  [343] = "19.57,-101.88,1.00,-90.00,-68.25,0.00,0,"
  [344] = "19.49,-101.70,1.00,-90.00,-68.30,0.00,1,"
  [345] = "19.42,-101.51,1.00,-90.00,-68.34,0.00,0,"
  [346] = "19.35,-101.32,1.00,-90.00,-68.38,0.00,1,"
  [347] = "19.27,-101.14,1.00,-90.00,-68.42,0.00,0,"
  [348] = "19.20,-100.95,1.00,-90.00,-68.46,0.00,1,"
  [349] = "19.13,-100.77,1.00,-90.00,-68.50,0.00,0,"
  [350] = "19.05,-100.58,1.00,-90.00,-68.55,0.00,1,"
  [351] = "18.98,-100.39,1.00,-90.00,-68.59,0.00,0,"
  [352] = "18.91,-100.21,1.00,-90.00,-68.63,0.00,1,"
  [353] = "18.83,-100.02,1.00,-90.00,-68.67,0.00,0,"
  [354] = "18.76,-99.83,1.00,-90.00,-68.71,0.00,1,"
  [355] = "18.69,-99.65,1.00,-90.00,-68.75,0.00,0,"
  [356] = "18.62,-99.46,1.00,-90.00,-68.80,0.00,1,"
  [357] = "18.54,-99.28,1.00,-90.00,-68.84,0.00,0,"
  [358] = "18.47,-99.09,1.00,-90.00,-68.88,0.00,1,"
  [359] = "18.40,-98.90,1.00,-90.00,-68.92,0.00,0,"
  [360] = "18.33,-98.72,1.00,-90.00,-68.96,0.00,1,"
  [361] = "18.26,-98.53,1.00,-90.00,-69.00,0.00,0,"
  [362] = "18.19,-98.34,1.00,-90.00,-69.05,0.00,1,"
  [363] = "18.11,-98.16,1.00,-90.00,-69.09,0.00,0,"
  [364] = "18.04,-97.97,1.00,-90.00,-69.13,0.00,1,"
  [365] = "17.97,-97.78,1.00,-90.00,-69.17,0.00,0,"
  [366] = "17.90,-97.59,1.00,-90.00,-69.21,0.00,1,"
  [367] = "17.83,-97.41,1.00,-90.00,-69.25,0.00,0,"
  [368] = "17.76,-97.22,1.00,-90.00,-69.30,0.00,1,"
  [369] = "17.69,-97.03,1.00,-90.00,-69.34,0.00,0,"
  [370] = "17.62,-96.85,1.00,-90.00,-69.38,0.00,1,"
  [371] = "17.55,-96.66,1.00,-90.00,-69.42,0.00,0,"
  [372] = "17.48,-96.47,1.00,-90.00,-69.46,0.00,1,"
  [373] = "17.41,-96.28,1.00,-90.00,-69.50,0.00,0,"
  [374] = "17.34,-96.10,1.00,-90.00,-69.55,0.00,1,"
  [375] = "17.27,-95.91,1.00,-90.00,-69.59,0.00,0,"
  [376] = "17.20,-95.72,1.00,-90.00,-69.63,0.00,1,"
  [377] = "17.13,-95.53,1.00,-90.00,-69.67,0.00,0,"
  [378] = "17.06,-95.35,1.00,-90.00,-69.71,0.00,1,"
  [379] = "16.99,-95.16,1.00,-90.00,-69.75,0.00,0,"
  [380] = "16.92,-94.97,1.00,-90.00,-69.80,0.00,1,"
  [381] = "16.85,-94.78,1.00,-90.00,-69.84,0.00,0,"
  [382] = "16.78,-94.60,1.00,-90.00,-69.88,0.00,1,"
  [383] = "16.71,-94.41,1.00,-90.00,-69.92,0.00,0,"
  [384] = "16.64,-94.22,1.00,-90.00,-69.96,0.00,1,"
  [385] = "16.58,-94.03,1.00,-90.00,-70.01,0.00,0,"
  [386] = "16.51,-93.84,1.00,-90.00,-70.05,0.00,1,"
  [387] = "16.44,-93.66,1.00,-90.00,-70.09,0.00,0,"
  [388] = "16.37,-93.47,1.00,-90.00,-70.13,0.00,1,"
  [389] = "16.30,-93.28,1.00,-90.00,-70.17,0.00,0,"
  [390] = "16.24,-93.09,1.00,-90.00,-70.21,0.00,1,"
  [391] = "16.17,-92.90,1.00,-90.00,-70.26,0.00,0,"
  [392] = "16.10,-92.72,1.00,-90.00,-70.30,0.00,1,"
  [393] = "16.03,-92.53,1.00,-90.00,-70.34,0.00,0,"
  [394] = "15.97,-92.34,1.00,-90.00,-70.38,0.00,1,"
  [395] = "15.90,-92.15,1.00,-90.00,-70.42,0.00,0,"
  [396] = "15.83,-91.96,1.00,-90.00,-70.46,0.00,1,"
  [397] = "15.77,-91.77,1.00,-90.00,-70.50,0.00,0,"
  [398] = "15.70,-91.59,1.00,-90.00,-70.55,0.00,1,"
  [399] = "15.63,-91.40,1.00,-90.00,-70.59,0.00,0,"
  [400] = "15.57,-91.21,1.00,-90.00,-70.63,0.00,1,"
  [401] = "15.50,-91.02,1.00,-90.00,-70.67,0.00,0,"
  [402] = "15.43,-90.83,1.00,-90.00,-70.71,0.00,1,"
  [403] = "15.37,-90.64,1.00,-90.00,-70.76,0.00,0,"
  [404] = "15.30,-90.45,1.00,-90.00,-70.80,0.00,1,"
  [405] = "15.24,-90.26,1.00,-90.00,-70.84,0.00,0,"
  [406] = "15.17,-90.08,1.00,-90.00,-70.88,0.00,1,"
  [407] = "15.10,-89.89,1.00,-90.00,-70.92,0.00,0,"
  [408] = "15.04,-89.70,1.00,-90.00,-70.96,0.00,1,"
  [409] = "14.97,-89.51,1.00,-90.00,-71.01,0.00,0,"
  [410] = "14.91,-89.32,1.00,-90.00,-71.05,0.00,1,"
  [411] = "14.84,-89.13,1.00,-90.00,-71.09,0.00,0,"
  [412] = "14.78,-88.94,1.00,-90.00,-71.13,0.00,1,"
  [413] = "14.72,-88.75,1.00,-90.00,-71.17,0.00,0,"
  [414] = "14.65,-88.56,1.00,-90.00,-71.21,0.00,1,"
  [415] = "14.59,-88.37,1.00,-90.00,-71.26,0.00,0,"
  [416] = "14.52,-88.18,1.00,-90.00,-71.30,0.00,1,"
  [417] = "14.46,-87.99,1.00,-90.00,-71.34,0.00,0,"
  [418] = "14.39,-87.80,1.00,-90.00,-71.38,0.00,1,"
  [419] = "14.33,-87.61,1.00,-90.00,-71.42,0.00,0,"
  [420] = "14.27,-87.43,1.00,-90.00,-71.46,0.00,1,"
  [421] = "14.20,-87.24,1.00,-90.00,-71.51,0.00,0,"
  [422] = "14.14,-87.05,1.00,-90.00,-71.55,0.00,1,"
  [423] = "14.08,-86.86,1.00,-90.00,-71.59,0.00,0,"
  [424] = "14.01,-86.67,1.00,-90.00,-71.63,0.00,1,"
  [425] = "13.95,-86.48,1.00,-90.00,-71.67,0.00,0,"
  [426] = "13.89,-86.29,1.00,-90.00,-71.71,0.00,1,"
  [427] = "13.82,-86.10,1.00,-90.00,-71.76,0.00,0,"
  [428] = "13.76,-85.91,1.00,-90.00,-71.80,0.00,1,"
  [429] = "13.70,-85.72,1.00,-90.00,-71.84,0.00,0,"
  [430] = "13.64,-85.53,1.00,-90.00,-71.88,0.00,1,"
  [431] = "13.58,-85.34,1.00,-90.00,-71.92,0.00,0,"
  [432] = "13.51,-85.15,1.00,-90.00,-71.96,0.00,1,"
  [433] = "13.45,-84.96,1.00,-90.00,-72.01,0.00,0,"
  [434] = "13.39,-84.77,1.00,-90.00,-72.05,0.00,1,"
  [435] = "13.33,-84.58,1.00,-90.00,-72.09,0.00,0,"
  [436] = "13.27,-84.39,1.00,-90.00,-72.13,0.00,1,"
  [437] = "13.21,-84.19,1.00,-90.00,-72.17,0.00,0,"
  [438] = "13.14,-84.00,1.00,-90.00,-72.21,0.00,1,"
  [439] = "13.08,-83.81,1.00,-90.00,-72.26,0.00,0,"
  [440] = "13.02,-83.62,1.00,-90.00,-72.30,0.00,1,"
  [441] = "12.96,-83.43,1.00,-90.00,-72.34,0.00,0,"
  [442] = "12.90,-83.24,1.00,-90.00,-72.38,0.00,1,"
  [443] = "12.84,-83.05,1.00,-90.00,-72.42,0.00,0,"
  [444] = "12.78,-82.86,1.00,-90.00,-72.46,0.00,1,"
  [445] = "12.72,-82.67,1.00,-90.00,-72.51,0.00,0,"
  [446] = "12.66,-82.48,1.00,-90.00,-72.55,0.00,1,"
  [447] = "12.60,-82.29,1.00,-90.00,-72.59,0.00,0,"
  [448] = "12.54,-82.10,1.00,-90.00,-72.63,0.00,1,"
  [449] = "12.48,-81.91,1.00,-90.00,-72.67,0.00,0,"
  [450] = "12.42,-81.72,1.00,-90.00,-72.71,0.00,1,"
  [451] = "12.36,-81.52,1.00,-90.00,-72.76,0.00,0,"
  [452] = "12.30,-81.33,1.00,-90.00,-72.80,0.00,1,"
  [453] = "12.24,-81.14,1.00,-90.00,-72.84,0.00,0,"
  [454] = "12.18,-80.95,1.00,-90.00,-72.88,0.00,1,"
  [455] = "12.13,-80.76,1.00,-90.00,-72.92,0.00,0,"
  [456] = "12.07,-80.57,1.00,-90.00,-72.96,0.00,1,"
  [457] = "12.01,-80.38,1.00,-90.00,-73.01,0.00,0,"
  [458] = "11.95,-80.19,1.00,-90.00,-73.05,0.00,1,"
  [459] = "11.89,-80.00,1.00,-90.00,-73.09,0.00,0,"
  [460] = "11.83,-79.80,1.00,-90.00,-73.13,0.00,1,"
  [461] = "11.78,-79.61,1.00,-90.00,-73.17,0.00,0,"
  [462] = "11.72,-79.42,1.00,-90.00,-73.21,0.00,1,"
  [463] = "11.66,-79.23,1.00,-90.00,-73.26,0.00,0,"
  [464] = "11.60,-79.04,1.00,-90.00,-73.30,0.00,1,"
  [465] = "11.55,-78.85,1.00,-90.00,-73.34,0.00,0,"
  [466] = "11.49,-78.66,1.00,-90.00,-73.38,0.00,1,"
  [467] = "11.43,-78.46,1.00,-90.00,-73.42,0.00,0,"
  [468] = "11.37,-78.27,1.00,-90.00,-73.46,0.00,1,"
  [469] = "11.32,-78.08,1.00,-90.00,-73.51,0.00,0,"
  [470] = "11.26,-77.89,1.00,-90.00,-73.55,0.00,1,"
  [471] = "11.20,-77.70,1.00,-90.00,-73.59,0.00,0,"
  [472] = "11.15,-77.50,1.00,-90.00,-73.63,0.00,1,"
  [473] = "11.09,-77.31,1.00,-90.00,-73.67,0.00,0,"
  [474] = "11.04,-77.12,1.00,-90.00,-73.71,0.00,1,"
  [475] = "10.98,-76.93,1.00,-90.00,-73.76,0.00,0,"
  [476] = "10.92,-76.74,1.00,-90.00,-73.80,0.00,1,"
  [477] = "10.87,-76.54,1.00,-90.00,-73.84,0.00,0,"
  [478] = "10.81,-76.35,1.00,-90.00,-73.88,0.00,1,"
  [479] = "10.76,-76.16,1.00,-90.00,-73.92,0.00,0,"
  [480] = "10.70,-75.97,1.00,-90.00,-73.96,0.00,1,"
  [481] = "10.65,-75.78,1.00,-90.00,-74.01,0.00,0,"
  [482] = "10.59,-75.58,1.00,-90.00,-74.05,0.00,1,"
  [483] = "10.54,-75.39,1.00,-90.00,-74.09,0.00,0,"
  [484] = "10.48,-75.20,1.00,-90.00,-74.13,0.00,1,"
  [485] = "10.43,-75.01,1.00,-90.00,-74.17,0.00,0,"
  [486] = "10.37,-74.81,1.00,-90.00,-74.21,0.00,1,"
  [487] = "10.32,-74.62,1.00,-90.00,-74.26,0.00,0,"
  [488] = "10.26,-74.43,1.00,-90.00,-74.30,0.00,1,"
  [489] = "10.21,-74.24,1.00,-90.00,-74.34,0.00,0,"
  [490] = "10.16,-74.04,1.00,-90.00,-74.38,0.00,1,"
  [491] = "10.10,-73.85,1.00,-90.00,-74.42,0.00,0,"
  [492] = "10.05,-73.66,1.00,-90.00,-74.46,0.00,1,"
  [493] = "9.99,-73.47,1.00,-90.00,-74.51,0.00,0,"
  [494] = "9.94,-73.27,1.00,-90.00,-74.55,0.00,1,"
  [495] = "9.89,-73.08,1.00,-90.00,-74.59,0.00,0,"
  [496] = "9.84,-72.89,1.00,-90.00,-74.63,0.00,1,"
  [497] = "9.78,-72.69,1.00,-90.00,-74.67,0.00,0,"
  [498] = "9.73,-72.50,1.00,-90.00,-74.71,0.00,1,"
  [499] = "9.68,-72.31,1.00,-90.00,-74.76,0.00,0,"
  [500] = "9.62,-72.12,1.00,-90.00,-74.80,0.00,1,"
  [501] = "9.57,-71.92,1.00,-90.00,-74.84,0.00,0,"
  [502] = "9.52,-71.73,1.00,-90.00,-74.88,0.00,1,"
  [503] = "9.47,-71.54,1.00,-90.00,-74.92,0.00,0,"
  [504] = "9.42,-71.34,1.00,-90.00,-74.96,0.00,1,"
  [505] = "9.36,-71.15,1.00,-90.00,-75.01,0.00,0,"
  [506] = "9.31,-70.96,1.00,-90.00,-75.05,0.00,1,"
  [507] = "9.26,-70.76,1.00,-90.00,-75.09,0.00,0,"
  [508] = "9.21,-70.57,1.00,-90.00,-75.13,0.00,1,"
  [509] = "9.16,-70.38,1.00,-90.00,-75.17,0.00,0,"
  [510] = "9.11,-70.18,1.00,-90.00,-75.21,0.00,1,"
  [511] = "9.06,-69.99,1.00,-90.00,-75.26,0.00,0,"
  [512] = "9.00,-69.80,1.00,-90.00,-75.30,0.00,1,"
  [513] = "8.95,-69.60,1.00,-90.00,-75.34,0.00,0,"
  [514] = "8.90,-69.41,1.00,-90.00,-75.38,0.00,1,"
  [515] = "8.85,-69.22,1.00,-90.00,-75.42,0.00,0,"
  [516] = "8.80,-69.02,1.00,-90.00,-75.46,0.00,1,"
  [517] = "8.75,-68.83,1.00,-90.00,-75.51,0.00,0,"
  [518] = "8.70,-68.64,1.00,-90.00,-75.55,0.00,1,"
  [519] = "8.65,-68.44,1.00,-90.00,-75.59,0.00,0,"
  [520] = "8.60,-68.25,1.00,-90.00,-75.63,0.00,1,"
  [521] = "8.55,-68.05,1.00,-90.00,-75.67,0.00,0,"
  [522] = "8.50,-67.86,1.00,-90.00,-75.71,0.00,1,"
  [523] = "8.46,-67.67,1.00,-90.00,-75.76,0.00,0,"
  [524] = "8.41,-67.47,1.00,-90.00,-75.80,0.00,1,"
  [525] = "8.36,-67.28,1.00,-90.00,-75.84,0.00,0,"
  [526] = "8.31,-67.09,1.00,-90.00,-75.88,0.00,1,"
  [527] = "8.26,-66.89,1.00,-90.00,-75.92,0.00,0,"
  [528] = "8.21,-66.70,1.00,-90.00,-75.96,0.00,1,"
  [529] = "8.16,-66.50,1.00,-90.00,-76.01,0.00,0,"
  [530] = "8.11,-66.31,1.00,-90.00,-76.05,0.00,1,"
  [531] = "8.07,-66.11,1.00,-90.00,-76.09,0.00,0,"
  [532] = "8.02,-65.92,1.00,-90.00,-76.13,0.00,1,"
  [533] = "7.97,-65.73,1.00,-90.00,-76.17,0.00,0,"
  [534] = "7.92,-65.53,1.00,-90.00,-76.21,0.00,1,"
  [535] = "7.87,-65.34,1.00,-90.00,-76.26,0.00,0,"
  [536] = "7.83,-65.14,1.00,-90.00,-76.30,0.00,1,"
  [537] = "7.78,-64.95,1.00,-90.00,-76.34,0.00,0,"
  [538] = "7.73,-64.76,1.00,-90.00,-76.38,0.00,1,"
  [539] = "7.69,-64.56,1.00,-90.00,-76.42,0.00,0,"
  [540] = "7.64,-64.37,1.00,-90.00,-76.46,0.00,1,"
  [541] = "7.59,-64.17,1.00,-90.00,-76.51,0.00,0,"
  [542] = "7.55,-63.98,1.00,-90.00,-76.55,0.00,1,"
  [543] = "7.50,-63.78,1.00,-90.00,-76.59,0.00,0,"
  [544] = "7.45,-63.59,1.00,-90.00,-76.63,0.00,1,"
  [545] = "7.41,-63.39,1.00,-90.00,-76.67,0.00,0,"
  [546] = "7.36,-63.20,1.00,-90.00,-76.71,0.00,1,"
  [547] = "7.31,-63.00,1.00,-90.00,-76.76,0.00,0,"
  [548] = "7.27,-62.81,1.00,-90.00,-76.80,0.00,1,"
  [549] = "7.22,-62.61,1.00,-90.00,-76.84,0.00,0,"
  [550] = "7.18,-62.42,1.00,-90.00,-76.88,0.00,1,"
  [551] = "7.13,-62.23,1.00,-90.00,-76.92,0.00,0,"
  [552] = "7.09,-62.03,1.00,-90.00,-76.96,0.00,1,"
  [553] = "7.04,-61.84,1.00,-90.00,-77.01,0.00,0,"
  [554] = "7.00,-61.64,1.00,-90.00,-77.05,0.00,1,"
  [555] = "6.95,-61.45,1.00,-90.00,-77.09,0.00,0,"
  [556] = "6.91,-61.25,1.00,-90.00,-77.13,0.00,1,"
  [557] = "6.86,-61.06,1.00,-90.00,-77.17,0.00,0,"
  [558] = "6.82,-60.86,1.00,-90.00,-77.21,0.00,1,"
  [559] = "6.77,-60.67,1.00,-90.00,-77.26,0.00,0,"
  [560] = "6.73,-60.47,1.00,-90.00,-77.30,0.00,1,"
  [561] = "6.69,-60.28,1.00,-90.00,-77.34,0.00,0,"
  [562] = "6.64,-60.08,1.00,-90.00,-77.38,0.00,1,"
  [563] = "6.60,-59.89,1.00,-90.00,-77.42,0.00,0,"
  [564] = "6.56,-59.69,1.00,-90.00,-77.46,0.00,1,"
  [565] = "6.51,-59.49,1.00,-90.00,-77.51,0.00,0,"
  [566] = "6.47,-59.30,1.00,-90.00,-77.55,0.00,1,"
  [567] = "6.43,-59.10,1.00,-90.00,-77.59,0.00,0,"
  [568] = "6.38,-58.91,1.00,-90.00,-77.63,0.00,1,"
  [569] = "6.34,-58.71,1.00,-90.00,-77.67,0.00,0,"
  [570] = "6.30,-58.52,1.00,-90.00,-77.71,0.00,1,"
  [571] = "6.26,-58.32,1.00,-90.00,-77.76,0.00,0,"
  [572] = "6.21,-58.13,1.00,-90.00,-77.80,0.00,1,"
  [573] = "6.17,-57.93,1.00,-90.00,-77.84,0.00,0,"
  [574] = "6.13,-57.74,1.00,-90.00,-77.88,0.00,1,"
  [575] = "6.09,-57.54,1.00,-90.00,-77.92,0.00,0,"
  [576] = "6.05,-57.35,1.00,-90.00,-77.96,0.00,1,"
  [577] = "6.00,-57.15,1.00,-90.00,-78.01,0.00,0,"
  [578] = "5.96,-56.95,1.00,-90.00,-78.05,0.00,1,"
  [579] = "5.92,-56.76,1.00,-90.00,-78.09,0.00,0,"
  [580] = "5.88,-56.56,1.00,-90.00,-78.13,0.00,1,"
  [581] = "5.84,-56.37,1.00,-90.00,-78.17,0.00,0,"
  [582] = "5.80,-56.17,1.00,-90.00,-78.21,0.00,1,"
  [583] = "5.76,-55.98,1.00,-90.00,-78.26,0.00,0,"
  [584] = "5.72,-55.78,1.00,-90.00,-78.30,0.00,1,"
  [585] = "5.68,-55.58,1.00,-90.00,-78.34,0.00,0,"
  [586] = "5.64,-55.39,1.00,-90.00,-78.38,0.00,1,"
  [587] = "5.60,-55.19,1.00,-90.00,-78.42,0.00,0,"
  [588] = "5.56,-55.00,1.00,-90.00,-78.46,0.00,1,"
  [589] = "5.52,-54.80,1.00,-90.00,-78.51,0.00,0,"
  [590] = "5.48,-54.60,1.00,-90.00,-78.55,0.00,1,"
  [591] = "5.44,-54.41,1.00,-90.00,-78.59,0.00,0,"
  [592] = "5.40,-54.21,1.00,-90.00,-78.63,0.00,1,"
  [593] = "5.36,-54.02,1.00,-90.00,-78.67,0.00,0,"
  [594] = "5.32,-53.82,1.00,-90.00,-78.71,0.00,1,"
  [595] = "5.28,-53.62,1.00,-90.00,-78.76,0.00,0,"
  [596] = "5.24,-53.43,1.00,-90.00,-78.80,0.00,1,"
  [597] = "5.20,-53.23,1.00,-90.00,-78.84,0.00,0,"
  [598] = "5.16,-53.03,1.00,-90.00,-78.88,0.00,1,"
  [599] = "5.12,-52.84,1.00,-90.00,-78.92,0.00,0,"
  [600] = "5.09,-52.64,1.00,-90.00,-78.96,0.00,1,"
  [601] = "5.05,-52.45,1.00,-90.00,-79.01,0.00,0,"
  [602] = "5.01,-52.25,1.00,-90.00,-79.05,0.00,1,"
  [603] = "4.97,-52.05,1.00,-90.00,-79.09,0.00,0,"
  [604] = "4.93,-51.86,1.00,-90.00,-79.13,0.00,1,"
  [605] = "4.90,-51.66,1.00,-90.00,-79.17,0.00,0,"
  [606] = "4.86,-51.46,1.00,-90.00,-79.21,0.00,1,"
  [607] = "4.82,-51.27,1.00,-90.00,-79.26,0.00,0,"
  [608] = "4.78,-51.07,1.00,-90.00,-79.30,0.00,1,"
  [609] = "4.75,-50.87,1.00,-90.00,-79.34,0.00,0,"
  [610] = "4.71,-50.68,1.00,-90.00,-79.38,0.00,1,"
  [611] = "4.67,-50.48,1.00,-90.00,-79.42,0.00,0,"
  [612] = "4.64,-50.28,1.00,-90.00,-79.46,0.00,1,"
  [613] = "4.60,-50.09,1.00,-90.00,-79.51,0.00,0,"
  [614] = "4.56,-49.89,1.00,-90.00,-79.55,0.00,1,"
  [615] = "4.53,-49.69,1.00,-90.00,-79.59,0.00,0,"
  [616] = "4.49,-49.50,1.00,-90.00,-79.63,0.00,1,"
  [617] = "4.46,-49.30,1.00,-90.00,-79.67,0.00,0,"
  [618] = "4.42,-49.10,1.00,-90.00,-79.71,0.00,1,"
  [619] = "4.38,-48.91,1.00,-90.00,-79.76,0.00,0,"
  [620] = "4.35,-48.71,1.00,-90.00,-79.80,0.00,1,"
  [621] = "4.31,-48.51,1.00,-90.00,-79.84,0.00,0,"
  [622] = "4.28,-48.32,1.00,-90.00,-79.88,0.00,1,"
  [623] = "4.24,-48.12,1.00,-90.00,-79.92,0.00,0,"
  [624] = "4.21,-47.92,1.00,-90.00,-79.96,0.00,1,"
  [625] = "4.17,-47.73,1.00,-90.00,-80.01,0.00,0,"
  [626] = "4.14,-47.53,1.00,-90.00,-80.05,0.00,1,"
  [627] = "4.10,-47.33,1.00,-90.00,-80.09,0.00,0,"
  [628] = "4.07,-47.14,1.00,-90.00,-80.13,0.00,1,"
  [629] = "4.04,-46.94,1.00,-90.00,-80.17,0.00,0,"
  [630] = "4.00,-46.74,1.00,-90.00,-80.21,0.00,1,"
  [631] = "3.97,-46.54,1.00,-90.00,-80.26,0.00,0,"
  [632] = "3.93,-46.35,1.00,-90.00,-80.30,0.00,1,"
  [633] = "3.90,-46.15,1.00,-90.00,-80.34,0.00,0,"
  [634] = "3.87,-45.95,1.00,-90.00,-80.38,0.00,1,"
  [635] = "3.83,-45.76,1.00,-90.00,-80.42,0.00,0,"
  [636] = "3.80,-45.56,1.00,-90.00,-80.46,0.00,1,"
  [637] = "3.77,-45.36,1.00,-90.00,-80.51,0.00,0,"
  [638] = "3.73,-45.16,1.00,-90.00,-80.55,0.00,1,"
  [639] = "3.70,-44.97,1.00,-90.00,-80.59,0.00,0,"
  [640] = "3.67,-44.77,1.00,-90.00,-80.63,0.00,1,"
  [641] = "3.64,-44.57,1.00,-90.00,-80.67,0.00,0,"
  [642] = "3.60,-44.37,1.00,-90.00,-80.71,0.00,1,"
  [643] = "3.57,-44.18,1.00,-90.00,-80.76,0.00,0,"
  [644] = "3.54,-43.98,1.00,-90.00,-80.80,0.00,1,"
  [645] = "3.51,-43.78,1.00,-90.00,-80.84,0.00,0,"
  [646] = "3.48,-43.58,1.00,-90.00,-80.88,0.00,1,"
  [647] = "3.44,-43.39,1.00,-90.00,-80.92,0.00,0,"
  [648] = "3.41,-43.19,1.00,-90.00,-80.96,0.00,1,"
  [649] = "3.38,-42.99,1.00,-90.00,-81.01,0.00,0,"
  [650] = "3.35,-42.79,1.00,-90.00,-81.05,0.00,1,"
  [651] = "3.32,-42.60,1.00,-90.00,-81.09,0.00,0,"
  [652] = "3.29,-42.40,1.00,-90.00,-81.13,0.00,1,"
  [653] = "3.26,-42.20,1.00,-90.00,-81.17,0.00,0,"
  [654] = "3.23,-42.00,1.00,-90.00,-81.21,0.00,1,"
  [655] = "3.20,-41.81,1.00,-90.00,-81.26,0.00,0,"
  [656] = "3.17,-41.61,1.00,-90.00,-81.30,0.00,1,"
  [657] = "3.14,-41.41,1.00,-90.00,-81.34,0.00,0,"
  [658] = "3.11,-41.21,1.00,-90.00,-81.38,0.00,1,"
  [659] = "3.08,-41.02,1.00,-90.00,-81.42,0.00,0,"
  [660] = "3.05,-40.82,1.00,-90.00,-81.46,0.00,1,"
  [661] = "3.02,-40.62,1.00,-90.00,-81.51,0.00,0,"
  [662] = "2.99,-40.42,1.00,-90.00,-81.55,0.00,1,"
  [663] = "2.96,-40.22,1.00,-90.00,-81.59,0.00,0,"
  [664] = "2.93,-40.03,1.00,-90.00,-81.63,0.00,1,"
  [665] = "2.90,-39.83,1.00,-90.00,-81.67,0.00,0,"
  [666] = "2.87,-39.63,1.00,-90.00,-81.71,0.00,1,"
  [667] = "2.84,-39.43,1.00,-90.00,-81.76,0.00,0,"
  [668] = "2.81,-39.23,1.00,-90.00,-81.80,0.00,1,"
  [669] = "2.78,-39.04,1.00,-90.00,-81.84,0.00,0,"
  [670] = "2.76,-38.84,1.00,-90.00,-81.88,0.00,1,"
  [671] = "2.73,-38.64,1.00,-90.00,-81.92,0.00,0,"
  [672] = "2.70,-38.44,1.00,-90.00,-81.96,0.00,1,"
  [673] = "2.67,-38.24,1.00,-90.00,-82.01,0.00,0,"
  [674] = "2.64,-38.05,1.00,-90.00,-82.05,0.00,1,"
  [675] = "2.62,-37.85,1.00,-90.00,-82.09,0.00,0,"
  [676] = "2.59,-37.65,1.00,-90.00,-82.13,0.00,1,"
  [677] = "2.56,-37.45,1.00,-90.00,-82.17,0.00,0,"
  [678] = "2.54,-37.25,1.00,-90.00,-82.21,0.00,1,"
  [679] = "2.51,-37.06,1.00,-90.00,-82.26,0.00,0,"
  [680] = "2.48,-36.86,1.00,-90.00,-82.30,0.00,1,"
  [681] = "2.45,-36.66,1.00,-90.00,-82.34,0.00,0,"
  [682] = "2.43,-36.46,1.00,-90.00,-82.38,0.00,1,"
  [683] = "2.40,-36.26,1.00,-90.00,-82.42,0.00,0,"
  [684] = "2.38,-36.06,1.00,-90.00,-82.46,0.00,1,"
  [685] = "2.35,-35.87,1.00,-90.00,-82.51,0.00,0,"
  [686] = "2.32,-35.67,1.00,-90.00,-82.55,0.00,1,"
  [687] = "2.30,-35.47,1.00,-90.00,-82.59,0.00,0,"
  [688] = "2.27,-35.27,1.00,-90.00,-82.63,0.00,1,"
  [689] = "2.25,-35.07,1.00,-90.00,-82.67,0.00,0,"
  [690] = "2.22,-34.87,1.00,-90.00,-82.71,0.00,1,"
  [691] = "2.20,-34.68,1.00,-90.00,-82.76,0.00,0,"
  [692] = "2.17,-34.48,1.00,-90.00,-82.80,0.00,1,"
  [693] = "2.14,-34.28,1.00,-90.00,-82.84,0.00,0,"
  [694] = "2.12,-34.08,1.00,-90.00,-82.88,0.00,1,"
  [695] = "2.10,-33.88,1.00,-90.00,-82.92,0.00,0,"
  [696] = "2.07,-33.68,1.00,-90.00,-82.96,0.00,1,"
  [697] = "2.05,-33.49,1.00,-90.00,-83.01,0.00,0,"
  [698] = "2.02,-33.29,1.00,-90.00,-83.05,0.00,1,"
  [699] = "2.00,-33.09,1.00,-90.00,-83.09,0.00,0,"
  [700] = "1.97,-32.89,1.00,-90.00,-83.13,0.00,1,"
  [701] = "1.95,-32.69,1.00,-90.00,-83.17,0.00,0,"
  [702] = "1.93,-32.49,1.00,-90.00,-83.21,0.00,1,"
  [703] = "1.90,-32.29,1.00,-90.00,-83.26,0.00,0,"
  [704] = "1.88,-32.10,1.00,-90.00,-83.30,0.00,1,"
  [705] = "1.86,-31.90,1.00,-90.00,-83.34,0.00,0,"
  [706] = "1.83,-31.70,1.00,-90.00,-83.38,0.00,1,"
  [707] = "1.81,-31.50,1.00,-90.00,-83.42,0.00,0,"
  [708] = "1.79,-31.30,1.00,-90.00,-83.46,0.00,1,"
  [709] = "1.76,-31.10,1.00,-90.00,-83.51,0.00,0,"
  [710] = "1.74,-30.90,1.00,-90.00,-83.55,0.00,1,"
  [711] = "1.72,-30.70,1.00,-90.00,-83.59,0.00,0,"
  [712] = "1.70,-30.51,1.00,-90.00,-83.63,0.00,1,"
  [713] = "1.68,-30.31,1.00,-90.00,-83.67,0.00,0,"
  [714] = "1.65,-30.11,1.00,-90.00,-83.71,0.00,1,"
  [715] = "1.63,-29.91,1.00,-90.00,-83.76,0.00,0,"
  [716] = "1.61,-29.71,1.00,-90.00,-83.80,0.00,1,"
  [717] = "1.59,-29.51,1.00,-90.00,-83.84,0.00,0,"
  [718] = "1.57,-29.31,1.00,-90.00,-83.88,0.00,1,"
  [719] = "1.55,-29.11,1.00,-90.00,-83.92,0.00,0,"
  [720] = "1.52,-28.92,1.00,-90.00,-83.96,0.00,1,"
  [721] = "1.50,-28.72,1.00,-90.00,-84.01,0.00,0,"
  [722] = "1.48,-28.52,1.00,-90.00,-84.05,0.00,1,"
  [723] = "1.46,-28.32,1.00,-90.00,-84.09,0.00,0,"
  [724] = "1.44,-28.12,1.00,-90.00,-84.13,0.00,1,"
  [725] = "1.42,-27.92,1.00,-90.00,-84.17,0.00,0,"
  [726] = "1.40,-27.72,1.00,-90.00,-84.21,0.00,1,"
  [727] = "1.38,-27.52,1.00,-90.00,-84.26,0.00,0,"
  [728] = "1.36,-27.32,1.00,-90.00,-84.30,0.00,1,"
  [729] = "1.34,-27.12,1.00,-90.00,-84.34,0.00,0,"
  [730] = "1.32,-26.93,1.00,-90.00,-84.38,0.00,1,"
  [731] = "1.30,-26.73,1.00,-90.00,-84.42,0.00,0,"
  [732] = "1.28,-26.53,1.00,-90.00,-84.46,0.00,1,"
  [733] = "1.26,-26.33,1.00,-90.00,-84.51,0.00,0,"
  [734] = "1.24,-26.13,1.00,-90.00,-84.55,0.00,1,"
  [735] = "1.23,-25.93,1.00,-90.00,-84.59,0.00,0,"
  [736] = "1.21,-25.73,1.00,-90.00,-84.63,0.00,1,"
  [737] = "1.19,-25.53,1.00,-90.00,-84.67,0.00,0,"
  [738] = "1.17,-25.33,1.00,-90.00,-84.71,0.00,1,"
  [739] = "1.15,-25.13,1.00,-90.00,-84.76,0.00,0,"
  [740] = "1.13,-24.93,1.00,-90.00,-84.80,0.00,1,"
  [741] = "1.11,-24.74,1.00,-90.00,-84.84,0.00,0,"
  [742] = "1.10,-24.54,1.00,-90.00,-84.88,0.00,1,"
  [743] = "1.08,-24.34,1.00,-90.00,-84.92,0.00,0,"
  [744] = "1.06,-24.14,1.00,-90.00,-84.96,0.00,1,"
  [745] = "1.04,-23.94,1.00,-90.00,-85.01,0.00,0,"
  [746] = "1.03,-23.74,1.00,-90.00,-85.05,0.00,1,"
  [747] = "1.01,-23.54,1.00,-90.00,-85.09,0.00,0,"
  [748] = "0.99,-23.34,1.00,-90.00,-85.13,0.00,1,"
  [749] = "0.98,-23.14,1.00,-90.00,-85.17,0.00,0,"
  [750] = "0.96,-22.94,1.00,-90.00,-85.21,0.00,1,"
  [751] = "0.94,-22.74,1.00,-90.00,-85.26,0.00,0,"
  [752] = "0.93,-22.54,1.00,-90.00,-85.30,0.00,1,"
  [753] = "0.91,-22.34,1.00,-90.00,-85.34,0.00,0,"
  [754] = "0.89,-22.14,1.00,-90.00,-85.38,0.00,1,"
  [755] = "0.88,-21.95,1.00,-90.00,-85.42,0.00,0,"
  [756] = "0.86,-21.75,1.00,-90.00,-85.46,0.00,1,"
  [757] = "0.85,-21.55,1.00,-90.00,-85.51,0.00,0,"
  [758] = "0.83,-21.35,1.00,-90.00,-85.55,0.00,1,"
  [759] = "0.81,-21.15,1.00,-90.00,-85.59,0.00,0,"
  [760] = "0.80,-20.95,1.00,-90.00,-85.63,0.00,1,"
  [761] = "0.78,-20.75,1.00,-90.00,-85.67,0.00,0,"
  [762] = "0.77,-20.55,1.00,-90.00,-85.71,0.00,1,"
  [763] = "0.75,-20.35,1.00,-90.00,-85.76,0.00,0,"
  [764] = "0.74,-20.15,1.00,-90.00,-85.80,0.00,1,"
  [765] = "0.72,-19.95,1.00,-90.00,-85.84,0.00,0,"
  [766] = "0.71,-19.75,1.00,-90.00,-85.88,0.00,1,"
  [767] = "0.70,-19.55,1.00,-90.00,-85.92,0.00,0,"
  [768] = "0.68,-19.35,1.00,-90.00,-85.96,0.00,1,"
  [769] = "0.67,-19.15,1.00,-90.00,-86.01,0.00,0,"
  [770] = "0.65,-18.95,1.00,-90.00,-86.05,0.00,1,"
  [771] = "0.64,-18.75,1.00,-90.00,-86.09,0.00,0,"
  [772] = "0.63,-18.55,1.00,-90.00,-86.13,0.00,1,"
  [773] = "0.61,-18.36,1.00,-90.00,-86.17,0.00,0,"
  [774] = "0.60,-18.16,1.00,-90.00,-86.21,0.00,1,"
  [775] = "0.59,-17.96,1.00,-90.00,-86.26,0.00,0,"
  [776] = "0.57,-17.76,1.00,-90.00,-86.30,0.00,1,"
  [777] = "0.56,-17.56,1.00,-90.00,-86.34,0.00,0,"
  [778] = "0.55,-17.36,1.00,-90.00,-86.38,0.00,1,"
  [779] = "0.54,-17.16,1.00,-90.00,-86.42,0.00,0,"
  [780] = "0.52,-16.96,1.00,-90.00,-86.46,0.00,1,"
  [781] = "0.51,-16.76,1.00,-90.00,-86.51,0.00,0,"
  [782] = "0.50,-16.56,1.00,-90.00,-86.55,0.00,1,"
  [783] = "0.49,-16.36,1.00,-90.00,-86.59,0.00,0,"
  [784] = "0.48,-16.16,1.00,-90.00,-86.63,0.00,1,"
  [785] = "0.46,-15.96,1.00,-90.00,-86.67,0.00,0,"
  [786] = "0.45,-15.76,1.00,-90.00,-86.71,0.00,1,"
  [787] = "0.44,-15.56,1.00,-90.00,-86.76,0.00,0,"
  [788] = "0.43,-15.36,1.00,-90.00,-86.80,0.00,1,"
  [789] = "0.42,-15.16,1.00,-90.00,-86.84,0.00,0,"
  [790] = "0.41,-14.96,1.00,-90.00,-86.88,0.00,1,"
  [791] = "0.40,-14.76,1.00,-90.00,-86.92,0.00,0,"
  [792] = "0.39,-14.56,1.00,-90.00,-86.96,0.00,1,"
  [793] = "0.38,-14.36,1.00,-90.00,-87.01,0.00,0,"
  [794] = "0.36,-14.16,1.00,-90.00,-87.05,0.00,1,"
  [795] = "0.35,-13.96,1.00,-90.00,-87.09,0.00,0,"
  [796] = "0.34,-13.76,1.00,-90.00,-87.13,0.00,1,"
  [797] = "0.33,-13.56,1.00,-90.00,-87.17,0.00,0,"
  [798] = "0.32,-13.36,1.00,-90.00,-87.21,0.00,1,"
  [799] = "0.32,-13.16,1.00,-90.00,-87.26,0.00,0,"
  [800] = "0.31,-12.96,1.00,-90.00,-87.30,0.00,1,"
  [801] = "0.30,-12.76,1.00,-90.00,-87.34,0.00,0,"
  [802] = "0.29,-12.56,1.00,-90.00,-87.38,0.00,1,"
  [803] = "0.28,-12.36,1.00,-90.00,-87.42,0.00,0,"
  [804] = "0.27,-12.17,1.00,-90.00,-87.46,0.00,1,"
  [805] = "0.26,-11.97,1.00,-90.00,-87.51,0.00,0,"
  [806] = "0.25,-11.77,1.00,-90.00,-87.55,0.00,1,"
  [807] = "0.24,-11.57,1.00,-90.00,-87.59,0.00,0,"
  [808] = "0.23,-11.37,1.00,-90.00,-87.63,0.00,1,"
  [809] = "0.23,-11.17,1.00,-90.00,-87.67,0.00,0,"
  [810] = "0.22,-10.97,1.00,-90.00,-87.71,0.00,1,"
  [811] = "0.21,-10.77,1.00,-90.00,-87.76,0.00,0,"
  [812] = "0.20,-10.57,1.00,-90.00,-87.80,0.00,1,"
  [813] = "0.20,-10.37,1.00,-90.00,-87.84,0.00,0,"
  [814] = "0.19,-10.17,1.00,-90.00,-87.88,0.00,1,"
  [815] = "0.18,-9.97,1.00,-90.00,-87.92,0.00,0,"
  [816] = "0.17,-9.77,1.00,-90.00,-87.96,0.00,1,"
  [817] = "0.17,-9.57,1.00,-90.00,-88.01,0.00,0,"
  [818] = "0.16,-9.37,1.00,-90.00,-88.05,0.00,1,"
  [819] = "0.15,-9.17,1.00,-90.00,-88.09,0.00,0,"
  [820] = "0.15,-8.97,1.00,-90.00,-88.13,0.00,1,"
  [821] = "0.14,-8.77,1.00,-90.00,-88.17,0.00,0,"
  [822] = "0.13,-8.57,1.00,-90.00,-88.21,0.00,1,"
  [823] = "0.13,-8.37,1.00,-90.00,-88.26,0.00,0,"
  [824] = "0.12,-8.17,1.00,-90.00,-88.30,0.00,1,"
  [825] = "0.12,-7.97,1.00,-90.00,-88.34,0.00,0,"
  [826] = "0.11,-7.77,1.00,-90.00,-88.38,0.00,1,"
  [827] = "0.10,-7.57,1.00,-90.00,-88.42,0.00,0,"
  [828] = "0.10,-7.37,1.00,-90.00,-88.46,0.00,1,"
  [829] = "0.09,-7.17,1.00,-90.00,-88.51,0.00,0,"
  [830] = "0.09,-6.97,1.00,-90.00,-88.55,0.00,1,"
  [831] = "0.08,-6.77,1.00,-90.00,-88.59,0.00,0,"
  [832] = "0.08,-6.57,1.00,-90.00,-88.63,0.00,1,"
  [833] = "0.07,-6.37,1.00,-90.00,-88.67,0.00,0,"
  [834] = "0.07,-6.17,1.00,-90.00,-88.71,0.00,1,"
  [835] = "0.06,-5.97,1.00,-90.00,-88.76,0.00,0,"
  [836] = "0.06,-5.77,1.00,-90.00,-88.80,0.00,1,"
  [837] = "0.06,-5.57,1.00,-90.00,-88.84,0.00,0,"
  [838] = "0.05,-5.37,1.00,-90.00,-88.88,0.00,1,"
  [839] = "0.05,-5.17,1.00,-90.00,-88.92,0.00,0,"
  [840] = "0.04,-4.97,1.00,-90.00,-88.96,0.00,1,"
  [841] = "0.04,-4.77,1.00,-90.00,-89.01,0.00,0,"
  [842] = "0.04,-4.57,1.00,-90.00,-89.05,0.00,1,"
  [843] = "0.03,-4.37,1.00,-90.00,-89.09,0.00,0,"
  [844] = "0.03,-4.17,1.00,-90.00,-89.13,0.00,1,"
  [845] = "0.03,-3.97,1.00,-90.00,-89.17,0.00,0,"
  [846] = "0.03,-3.77,1.00,-90.00,-89.21,0.00,1,"
  [847] = "0.02,-3.57,1.00,-90.00,-89.26,0.00,0,"
  [848] = "0.02,-3.37,1.00,-90.00,-89.30,0.00,1,"
  [849] = "0.02,-3.17,1.00,-90.00,-89.34,0.00,0,"
  [850] = "0.02,-2.97,1.00,-90.00,-89.38,0.00,1,"
  [851] = "0.01,-2.77,1.00,-90.00,-89.42,0.00,0,"
  [852] = "0.01,-2.57,1.00,-90.00,-89.46,0.00,1,"
  [853] = "0.01,-2.37,1.00,-90.00,-89.51,0.00,0,"
  [854] = "0.01,-2.17,1.00,-90.00,-89.55,0.00,1,"
  [855] = "0.01,-1.97,1.00,-90.00,-89.59,0.00,0,"
  [856] = "0.01,-1.77,1.00,-90.00,-89.63,0.00,1,"
  [857] = "0.00,-1.57,1.00,-90.00,-89.67,0.00,0,"
  [858] = "0.00,-1.37,1.00,-90.00,-89.71,0.00,1,"
  [859] = "0.00,-1.17,1.00,-90.00,-89.76,0.00,0,"
  [860] = "0.00,-0.97,1.00,-90.00,-89.80,0.00,1,"
  [861] = "0.00,-0.77,1.00,-90.00,-89.84,0.00,0,"
  [862] = "0.00,-0.57,1.00,-90.00,-89.88,0.00,1,"
  [863] = "0.00,-0.37,1.00,-90.00,-89.92,0.00,0,"
  [864] = "0.00,-0.17,1.00,-90.00,-89.96,0.00,1,"
  [865] = "0.00,0.03,1.00,90.00,89.99,0.00,0,"
  [866] = "0.00,0.23,1.00,90.00,89.95,0.00,1,"
  [867] = "0.00,0.43,1.00,90.00,89.91,0.00,0,"
  [868] = "0.00,0.63,1.00,90.00,89.87,0.00,1,"
  [869] = "0.00,0.83,1.00,90.00,89.83,0.00,0,"
  [870] = "0.00,1.03,1.00,90.00,89.79,0.00,1,"
  [871] = "0.00,1.23,1.00,90.00,89.74,0.00,0,"
  [872] = "0.00,1.43,1.00,90.00,89.70,0.00,1,"
  [873] = "0.00,1.63,1.00,90.00,89.66,0.00,0,"
  [874] = "0.01,1.83,1.00,90.00,89.62,0.00,1,"
  [875] = "0.01,2.03,1.00,90.00,89.58,0.00,0,"
  [876] = "0.01,2.23,1.00,90.00,89.54,0.00,1,"
  [877] = "0.01,2.43,1.00,90.00,89.49,0.00,0,"
  [878] = "0.01,2.63,1.00,90.00,89.45,0.00,1,"
  [879] = "0.01,2.83,1.00,90.00,89.41,0.00,0,"
  [880] = "0.02,3.03,1.00,90.00,89.37,0.00,1,"
  [881] = "0.02,3.23,1.00,90.00,89.33,0.00,0,"
  [882] = "0.02,3.43,1.00,90.00,89.29,0.00,1,"
  [883] = "0.02,3.63,1.00,90.00,89.24,0.00,0,"
  [884] = "0.03,3.83,1.00,90.00,89.20,0.00,1,"
  [885] = "0.03,4.03,1.00,90.00,89.16,0.00,0,"
  [886] = "0.03,4.23,1.00,90.00,89.12,0.00,1,"
  [887] = "0.04,4.43,1.00,90.00,89.08,0.00,0,"
  [888] = "0.04,4.63,1.00,90.00,89.04,0.00,1,"
  [889] = "0.04,4.83,1.00,90.00,88.99,0.00,0,"
  [890] = "0.05,5.03,1.00,90.00,88.95,0.00,1,"
  [891] = "0.05,5.23,1.00,90.00,88.91,0.00,0,"
  [892] = "0.05,5.43,1.00,90.00,88.87,0.00,1,"
  [893] = "0.06,5.63,1.00,90.00,88.83,0.00,0,"
  [894] = "0.06,5.83,1.00,90.00,88.79,0.00,1,"
  [895] = "0.07,6.03,1.00,90.00,88.74,0.00,0,"
  [896] = "0.07,6.23,1.00,90.00,88.70,0.00,1,"
  [897] = "0.08,6.43,1.00,90.00,88.66,0.00,0,"
  [898] = "0.08,6.63,1.00,90.00,88.62,0.00,1,"
  [899] = "0.08,6.83,1.00,90.00,88.58,0.00,0,"
  [900] = "0.09,7.03,1.00,90.00,88.54,0.00,1,"
  [901] = "0.10,7.23,1.00,90.00,88.49,0.00,0,"
  [902] = "0.10,7.43,1.00,90.00,88.45,0.00,1,"
  [903] = "0.11,7.63,1.00,90.00,88.41,0.00,0,"
  [904] = "0.11,7.83,1.00,90.00,88.37,0.00,1,"
  [905] = "0.12,8.03,1.00,90.00,88.33,0.00,0,"
  [906] = "0.12,8.23,1.00,90.00,88.29,0.00,1,"
  [907] = "0.13,8.43,1.00,90.00,88.24,0.00,0,"
  [908] = "0.14,8.63,1.00,90.00,88.20,0.00,1,"
  [909] = "0.14,8.83,1.00,90.00,88.16,0.00,0,"
  [910] = "0.15,9.03,1.00,90.00,88.12,0.00,1,"
  [911] = "0.15,9.23,1.00,90.00,88.08,0.00,0,"
  [912] = "0.16,9.43,1.00,90.00,88.04,0.00,1,"
  [913] = "0.17,9.63,1.00,90.00,87.99,0.00,0,"
  [914] = "0.18,9.83,1.00,90.00,87.95,0.00,1,"
  [915] = "0.18,10.03,1.00,90.00,87.91,0.00,0,"
  [916] = "0.19,10.23,1.00,90.00,87.87,0.00,1,"
  [917] = "0.20,10.43,1.00,90.00,87.83,0.00,0,"
  [918] = "0.21,10.63,1.00,90.00,87.79,0.00,1,"
  [919] = "0.21,10.83,1.00,90.00,87.74,0.00,0,"
  [920] = "0.22,11.03,1.00,90.00,87.70,0.00,1,"
  [921] = "0.23,11.23,1.00,90.00,87.66,0.00,0,"
  [922] = "0.24,11.43,1.00,90.00,87.62,0.00,1,"
  [923] = "0.25,11.63,1.00,90.00,87.58,0.00,0,"
  [924] = "0.25,11.83,1.00,90.00,87.53,0.00,1,"
  [925] = "0.26,12.03,1.00,90.00,87.49,0.00,0,"
  [926] = "0.27,12.23,1.00,90.00,87.45,0.00,1,"
  [927] = "0.28,12.43,1.00,90.00,87.41,0.00,0,"
  [928] = "0.29,12.63,1.00,90.00,87.37,0.00,1,"
  [929] = "0.30,12.83,1.00,90.00,87.33,0.00,0,"
  [930] = "0.31,13.03,1.00,90.00,87.28,0.00,1,"
  [931] = "0.32,13.23,1.00,90.00,87.24,0.00,0,"
  [932] = "0.33,13.43,1.00,90.00,87.20,0.00,1,"
  [933] = "0.34,13.63,1.00,90.00,87.16,0.00,0,"
  [934] = "0.35,13.83,1.00,90.00,87.12,0.00,1,"
  [935] = "0.36,14.02,1.00,90.00,87.08,0.00,0,"
  [936] = "0.37,14.22,1.00,90.00,87.03,0.00,1,"
  [937] = "0.38,14.42,1.00,90.00,86.99,0.00,0,"
  [938] = "0.39,14.62,1.00,90.00,86.95,0.00,1,"
  [939] = "0.40,14.82,1.00,90.00,86.91,0.00,0,"
  [940] = "0.41,15.02,1.00,90.00,86.87,0.00,1,"
  [941] = "0.42,15.22,1.00,90.00,86.83,0.00,0,"
  [942] = "0.43,15.42,1.00,90.00,86.78,0.00,1,"
  [943] = "0.44,15.62,1.00,90.00,86.74,0.00,0,"
  [944] = "0.46,15.82,1.00,90.00,86.70,0.00,1,"
  [945] = "0.47,16.02,1.00,90.00,86.66,0.00,0,"
  [946] = "0.48,16.22,1.00,90.00,86.62,0.00,1,"
  [947] = "0.49,16.42,1.00,90.00,86.58,0.00,0,"
  [948] = "0.50,16.62,1.00,90.00,86.53,0.00,1,"
  [949] = "0.51,16.82,1.00,90.00,86.49,0.00,0,"
  [950] = "0.53,17.02,1.00,90.00,86.45,0.00,1,"
  [951] = "0.54,17.22,1.00,90.00,86.41,0.00,0,"
  [952] = "0.55,17.42,1.00,90.00,86.37,0.00,1,"
  [953] = "0.56,17.62,1.00,90.00,86.33,0.00,0,"
  [954] = "0.58,17.82,1.00,90.00,86.28,0.00,1,"
  [955] = "0.59,18.02,1.00,90.00,86.24,0.00,0,"
  [956] = "0.60,18.22,1.00,90.00,86.20,0.00,1,"
  [957] = "0.62,18.42,1.00,90.00,86.16,0.00,0,"
  [958] = "0.63,18.62,1.00,90.00,86.12,0.00,1,"
  [959] = "0.64,18.82,1.00,90.00,86.08,0.00,0,"
  [960] = "0.66,19.02,1.00,90.00,86.03,0.00,1,"
  [961] = "0.67,19.22,1.00,90.00,85.99,0.00,0,"
  [962] = "0.69,19.41,1.00,90.00,85.95,0.00,1,"
  [963] = "0.70,19.61,1.00,90.00,85.91,0.00,0,"
  [964] = "0.71,19.81,1.00,90.00,85.87,0.00,1,"
  [965] = "0.73,20.01,1.00,90.00,85.83,0.00,0,"
  [966] = "0.74,20.21,1.00,90.00,85.78,0.00,1,"
  [967] = "0.76,20.41,1.00,90.00,85.74,0.00,0,"
  [968] = "0.77,20.61,1.00,90.00,85.70,0.00,1,"
  [969] = "0.79,20.81,1.00,90.00,85.66,0.00,0,"
  [970] = "0.80,21.01,1.00,90.00,85.62,0.00,1,"
  [971] = "0.82,21.21,1.00,90.00,85.58,0.00,0,"
  [972] = "0.83,21.41,1.00,90.00,85.53,0.00,1,"
  [973] = "0.85,21.61,1.00,90.00,85.49,0.00,0,"
  [974] = "0.87,21.81,1.00,90.00,85.45,0.00,1,"
  [975] = "0.88,22.01,1.00,90.00,85.41,0.00,0,"
  [976] = "0.90,22.21,1.00,90.00,85.37,0.00,1,"
  [977] = "0.91,22.41,1.00,90.00,85.33,0.00,0,"
  [978] = "0.93,22.61,1.00,90.00,85.28,0.00,1,"
  [979] = "0.95,22.80,1.00,90.00,85.24,0.00,0,"
  [980] = "0.96,23.00,1.00,90.00,85.20,0.00,1,"
  [981] = "0.98,23.20,1.00,90.00,85.16,0.00,0,"
  [982] = "1.00,23.40,1.00,90.00,85.12,0.00,1,"
  [983] = "1.01,23.60,1.00,90.00,85.08,0.00,0,"
  [984] = "1.03,23.80,1.00,90.00,85.03,0.00,1,"
  [985] = "1.05,24.00,1.00,90.00,84.99,0.00,0,"
  [986] = "1.07,24.20,1.00,90.00,84.95,0.00,1,"
  [987] = "1.08,24.40,1.00,90.00,84.91,0.00,0,"
  [988] = "1.10,24.60,1.00,90.00,84.87,0.00,1,"
  [989] = "1.12,24.80,1.00,90.00,84.83,0.00,0,"
  [990] = "1.14,25.00,1.00,90.00,84.78,0.00,1,"
  [991] = "1.16,25.20,1.00,90.00,84.74,0.00,0,"
  [992] = "1.18,25.39,1.00,90.00,84.70,0.00,1,"
  [993] = "1.19,25.59,1.00,90.00,84.66,0.00,0,"
  [994] = "1.21,25.79,1.00,90.00,84.62,0.00,1,"
  [995] = "1.23,25.99,1.00,90.00,84.58,0.00,0,"
  [996] = "1.25,26.19,1.00,90.00,84.53,0.00,1,"
  [997] = "1.27,26.39,1.00,90.00,84.49,0.00,0,"
  [998] = "1.29,26.59,1.00,90.00,84.45,0.00,1,"
  [999] = "1.31,26.79,1.00,90.00,84.41,0.00,0,"
string sTxtfile[511]
  [0] = "path0.txt"
  [1] = "path1.txt"
  [2] = "path2.txt"
  [3] = "path3.txt"
  [4] = "path4.txt"
  [5] = "path5.txt"
  [6] = "path6.txt"
  [7] = "path7.txt"
  [8] = "path8.txt"
  [9] = "path9.txt"
  [10] = "path10.txt"
  [11] = "path11.txt"
  [12] = "path12.txt"
  [13] = "path13.txt"
  [14] = "path14.txt"
  [15] = "path15.txt"
  [16] = "path16.txt"
  [17] = "path17.txt"
  [18] = "path18.txt"
  [19] = "path19.txt"
  [20] = "path20.txt"
  [21] = "path21.txt"
  [22] = "path22.txt"
  [23] = "path23.txt"
  [24] = "path24.txt"
  [25] = "path25.txt"
  [26] = "path26.txt"
  [27] = "path27.txt"
  [28] = "path28.txt"
  [29] = "path29.txt"
  [30] = "path30.txt"
  [31] = "path31.txt"
  [32] = "path32.txt"
  [33] = "path33.txt"
  [34] = "path34.txt"
  [35] = "path35.txt"
  [36] = "path36.txt"
  [37] = "path37.txt"
  [38] = "path38.txt"
  [39] = "path39.txt"
  [40] = "path40.txt"
  [41] = "path41.txt"
  [42] = "path42.txt"
  [43] = "path43.txt"
  [44] = "path44.txt"
  [45] = "path45.txt"
  [46] = "path46.txt"
  [47] = "path47.txt"
  [48] = "path48.txt"
  [49] = "path49.txt"
  [50] = "path50.txt"
  [51] = "path51.txt"
  [52] = "path52.txt"
  [53] = "path53.txt"
  [54] = "path54.txt"
  [55] = "path55.txt"
  [56] = "path56.txt"
  [57] = "path57.txt"
  [58] = "path58.txt"
  [59] = "path59.txt"
  [60] = "path60.txt"
  [61] = "path61.txt"
  [62] = "path62.txt"
  [63] = "path63.txt"
  [64] = "path64.txt"
  [65] = "path65.txt"
  [66] = "path66.txt"
  [67] = "path67.txt"
  [68] = "path68.txt"
  [69] = "path69.txt"
  [70] = "path70.txt"
  [71] = "path71.txt"
  [72] = "path72.txt"
  [73] = "path73.txt"
  [74] = "path74.txt"
  [75] = "path75.txt"
  [76] = "path76.txt"
  [77] = "path77.txt"
  [78] = "path78.txt"
  [79] = "path79.txt"
  [80] = "path80.txt"
  [81] = "path81.txt"
  [82] = "path82.txt"
  [83] = "path83.txt"
  [84] = "path84.txt"
  [85] = "path85.txt"
  [86] = "path86.txt"
  [87] = "path87.txt"
  [88] = "path88.txt"
  [89] = "path89.txt"
  [90] = "path90.txt"
  [91] = "path91.txt"
  [92] = "path92.txt"
  [93] = "path93.txt"
  [94] = "path94.txt"
  [95] = "path95.txt"
  [96] = "path96.txt"
  [97] = "path97.txt"
  [98] = "path98.txt"
  [99] = "path99.txt"
  [100] = "path100.txt"
  [101] = "path101.txt"
  [102] = "path102.txt"
  [103] = "path103.txt"
  [104] = "path104.txt"
  [105] = "path105.txt"
  [106] = "path106.txt"
  [107] = "path107.txt"
  [108] = "path108.txt"
  [109] = "path109.txt"
  [110] = "path110.txt"
  [111] = "path111.txt"
  [112] = "path112.txt"
  [113] = "path113.txt"
  [114] = "path114.txt"
  [115] = "path115.txt"
  [116] = "path116.txt"
  [117] = "path117.txt"
  [118] = "path118.txt"
  [119] = "path119.txt"
  [120] = "path120.txt"
  [121] = "path121.txt"
  [122] = "path122.txt"
  [123] = "path123.txt"
  [124] = "path124.txt"
  [125] = "path125.txt"
  [126] = "path126.txt"
  [127] = "path127.txt"
  [128] = "path128.txt"
  [129] = "path129.txt"
  [130] = "path130.txt"
  [131] = "path131.txt"
  [132] = "path132.txt"
  [133] = "path133.txt"
  [134] = "path134.txt"
  [135] = "path135.txt"
  [136] = "path136.txt"
  [137] = "path137.txt"
  [138] = "path138.txt"
  [139] = "path139.txt"
  [140] = "path140.txt"
  [141] = "path141.txt"
  [142] = "path142.txt"
  [143] = "path143.txt"
  [144] = "path144.txt"
  [145] = "path145.txt"
  [146] = "path146.txt"
  [147] = "path147.txt"
  [148] = "path148.txt"
  [149] = "path149.txt"
  [150] = "path150.txt"
  [151] = "path151.txt"
  [152] = "path152.txt"
  [153] = "path153.txt"
  [154] = "path154.txt"
  [155] = "path155.txt"
  [156] = "path156.txt"
  [157] = "path157.txt"
  [158] = "path158.txt"
  [159] = "path159.txt"
  [160] = "path160.txt"
  [161] = "path161.txt"
  [162] = "path162.txt"
  [163] = "path163.txt"
  [164] = "path164.txt"
  [165] = "path165.txt"
  [166] = "path166.txt"
  [167] = "path167.txt"
  [168] = "path168.txt"
  [169] = "path169.txt"
  [170] = "path170.txt"
  [171] = "path171.txt"
  [172] = "path172.txt"
  [173] = "path173.txt"
  [174] = "path174.txt"
  [175] = "path175.txt"
  [176] = "path176.txt"
  [177] = "path177.txt"
  [178] = "path178.txt"
  [179] = "path179.txt"
  [180] = "path180.txt"
  [181] = "path181.txt"
  [182] = "path182.txt"
  [183] = "path183.txt"
  [184] = "path184.txt"
  [185] = "path185.txt"
  [186] = "path186.txt"
  [187] = "path187.txt"
  [188] = "path188.txt"
  [189] = "path189.txt"
  [190] = "path190.txt"
  [191] = "path191.txt"
  [192] = "path192.txt"
  [193] = "path193.txt"
  [194] = "path194.txt"
  [195] = "path195.txt"
  [196] = "path196.txt"
  [197] = "path197.txt"
  [198] = "path198.txt"
  [199] = "path199.txt"
  [200] = "path200.txt"
  [201] = "path201.txt"
  [202] = "path202.txt"
  [203] = "path203.txt"
  [204] = "path204.txt"
  [205] = "path205.txt"
  [206] = "path206.txt"
  [207] = "path207.txt"
  [208] = "path208.txt"
  [209] = "path209.txt"
  [210] = "path210.txt"
  [211] = "path211.txt"
  [212] = "path212.txt"
  [213] = "path213.txt"
  [214] = "path214.txt"
  [215] = "path215.txt"
  [216] = "path216.txt"
  [217] = "path217.txt"
  [218] = "path218.txt"
  [219] = "path219.txt"
  [220] = "path220.txt"
  [221] = "path221.txt"
  [222] = "path222.txt"
  [223] = "path223.txt"
  [224] = "path224.txt"
  [225] = "path225.txt"
  [226] = "path226.txt"
  [227] = "path227.txt"
  [228] = "path228.txt"
  [229] = "path229.txt"
  [230] = "path230.txt"
  [231] = "path231.txt"
  [232] = "path232.txt"
  [233] = "path233.txt"
  [234] = "path234.txt"
  [235] = "path235.txt"
  [236] = "path236.txt"
  [237] = "path237.txt"
  [238] = "path238.txt"
  [239] = "path239.txt"
  [240] = "path240.txt"
  [241] = "path241.txt"
  [242] = "path242.txt"
  [243] = "path243.txt"
  [244] = "path244.txt"
  [245] = "path245.txt"
  [246] = "path246.txt"
  [247] = "path247.txt"
  [248] = "path248.txt"
  [249] = "path249.txt"
  [250] = "path250.txt"
  [251] = "path251.txt"
  [252] = "path252.txt"
  [253] = "path253.txt"
  [254] = "path254.txt"
  [255] = "path255.txt"
  [256] = "path256.txt"
  [257] = "path257.txt"
  [258] = "path258.txt"
  [259] = "path259.txt"
  [260] = "path260.txt"
  [261] = "path261.txt"
  [262] = "path262.txt"
  [263] = "path263.txt"
  [264] = "path264.txt"
  [265] = "path265.txt"
  [266] = "path266.txt"
  [267] = "path267.txt"
  [268] = "path268.txt"
  [269] = "path269.txt"
  [270] = "path270.txt"
  [271] = "path271.txt"
  [272] = "path272.txt"
  [273] = "path273.txt"
  [274] = "path274.txt"
  [275] = "path275.txt"
  [276] = "path276.txt"
  [277] = "path277.txt"
  [278] = "path278.txt"
  [279] = "path279.txt"
  [280] = "path280.txt"
  [281] = "path281.txt"
  [282] = "path282.txt"
  [283] = "path283.txt"
  [284] = "path284.txt"
  [285] = "path285.txt"
  [286] = "path286.txt"
  [287] = "path287.txt"
  [288] = "path288.txt"
  [289] = "path289.txt"
  [290] = "path290.txt"
  [291] = "path291.txt"
  [292] = "path292.txt"
  [293] = "path293.txt"
  [294] = "path294.txt"
  [295] = "path295.txt"
  [296] = "path296.txt"
  [297] = "path297.txt"
  [298] = "path298.txt"
  [299] = "path299.txt"
  [300] = "path300.txt"
  [301] = "path301.txt"
  [302] = "path302.txt"
  [303] = "path303.txt"
  [304] = "path304.txt"
  [305] = "path305.txt"
  [306] = "path306.txt"
  [307] = "path307.txt"
  [308] = "path308.txt"
  [309] = "path309.txt"
  [310] = "path310.txt"
  [311] = "path311.txt"
  [312] = "path312.txt"
  [313] = "path313.txt"
  [314] = "path314.txt"
  [315] = "path315.txt"
  [316] = "path316.txt"
  [317] = "path317.txt"
  [318] = "path318.txt"
  [319] = "path319.txt"
  [320] = "path320.txt"
  [321] = "path321.txt"
  [322] = "path322.txt"
  [323] = "path323.txt"
  [324] = "path324.txt"
  [325] = "path325.txt"
  [326] = "path326.txt"
  [327] = "path327.txt"
  [328] = "path328.txt"
  [329] = "path329.txt"
  [330] = "path330.txt"
  [331] = "path331.txt"
  [332] = "path332.txt"
  [333] = "path333.txt"
  [334] = "path334.txt"
  [335] = "path335.txt"
  [336] = "path336.txt"
  [337] = "path337.txt"
  [338] = "path338.txt"
  [339] = "path339.txt"
  [340] = "path340.txt"
  [341] = "path341.txt"
  [342] = "path342.txt"
  [343] = "path343.txt"
  [344] = "path344.txt"
  [345] = "path345.txt"
  [346] = "path346.txt"
  [347] = "path347.txt"
  [348] = "path348.txt"
  [349] = "path349.txt"
  [350] = "path350.txt"
  [351] = "path351.txt"
  [352] = "path352.txt"
  [353] = "path353.txt"
  [354] = "path354.txt"
  [355] = "path355.txt"
  [356] = "path356.txt"
  [357] = "path357.txt"
  [358] = "path358.txt"
  [359] = "path359.txt"
  [360] = "path360.txt"
  [361] = "path361.txt"
  [362] = "path362.txt"
  [363] = "path363.txt"
  [364] = "path364.txt"
  [365] = "path365.txt"
  [366] = "path366.txt"
  [367] = "path367.txt"
  [368] = "path368.txt"
  [369] = "path369.txt"
  [370] = "path370.txt"
  [371] = "path371.txt"
  [372] = "path372.txt"
  [373] = "path373.txt"
  [374] = "path374.txt"
  [375] = "path375.txt"
  [376] = "path376.txt"
  [377] = "path377.txt"
  [378] = "path378.txt"
  [379] = "path379.txt"
  [380] = "path380.txt"
  [381] = "path381.txt"
  [382] = "path382.txt"
  [383] = "path383.txt"
  [384] = "path384.txt"
  [385] = "path385.txt"
  [386] = "path386.txt"
  [387] = "path387.txt"
  [388] = "path388.txt"
  [389] = "path389.txt"
  [390] = "path390.txt"
  [391] = "path391.txt"
  [392] = "path392.txt"
  [393] = "path393.txt"
  [394] = "path394.txt"
  [395] = "path395.txt"
  [396] = "path396.txt"
  [397] = "path397.txt"
  [398] = "path398.txt"
  [399] = "path399.txt"
  [400] = "path400.txt"
  [401] = "path401.txt"
  [402] = "path402.txt"
  [403] = "path403.txt"
  [404] = "path404.txt"
  [405] = "path405.txt"
  [406] = "path406.txt"
  [407] = "path407.txt"
  [408] = "path408.txt"
  [409] = "path409.txt"
  [410] = "path410.txt"
  [411] = "path411.txt"
  [412] = "path412.txt"
  [413] = "path413.txt"
  [414] = "path414.txt"
  [415] = "path415.txt"
  [416] = "path416.txt"
  [417] = "path417.txt"
  [418] = "path418.txt"
  [419] = "path419.txt"
  [420] = "path420.txt"
  [421] = "path421.txt"
  [422] = "path422.txt"
  [423] = "path423.txt"
  [424] = "path424.txt"
  [425] = "path425.txt"
  [426] = "path426.txt"
  [427] = "path427.txt"
  [428] = "path428.txt"
  [429] = "path429.txt"
  [430] = "path430.txt"
  [431] = "path431.txt"
  [432] = "path432.txt"
  [433] = "path433.txt"
  [434] = "path434.txt"
  [435] = "path435.txt"
  [436] = "path436.txt"
  [437] = "path437.txt"
  [438] = "path438.txt"
  [439] = "path439.txt"
  [440] = "path440.txt"
  [441] = "path441.txt"
  [442] = "path442.txt"
  [443] = "path443.txt"
  [444] = "path444.txt"
  [445] = "path445.txt"
  [446] = "path446.txt"
  [447] = "path447.txt"
  [448] = "path448.txt"
  [449] = "path449.txt"
  [450] = "path450.txt"
  [451] = "path451.txt"
  [452] = "path452.txt"
  [453] = "path453.txt"
  [454] = "path454.txt"
  [455] = "path455.txt"
  [456] = "path456.txt"
  [457] = "path457.txt"
  [458] = "path458.txt"
  [459] = "path459.txt"
  [460] = "path460.txt"
  [461] = "path461.txt"
  [462] = "path462.txt"
  [463] = "path463.txt"
  [464] = "path464.txt"
  [465] = "path465.txt"
  [466] = "path466.txt"
  [467] = "path467.txt"
  [468] = "path468.txt"
  [469] = "path469.txt"
  [470] = "path470.txt"
  [471] = "path471.txt"
  [472] = "path472.txt"
  [473] = "path473.txt"
  [474] = "path474.txt"
  [475] = "path475.txt"
  [476] = "path476.txt"
  [477] = "path477.txt"
  [478] = "path478.txt"
  [479] = "path479.txt"
  [480] = "path480.txt"
  [481] = "path481.txt"
  [482] = "path482.txt"
  [483] = "path483.txt"
  [484] = "path484.txt"
  [485] = "path485.txt"
  [486] = "path486.txt"
  [487] = "path487.txt"
  [488] = "path488.txt"
  [489] = "path489.txt"
  [490] = "path490.txt"
  [491] = "path491.txt"
  [492] = "path492.txt"
  [493] = "path493.txt"
  [494] = "path494.txt"
  [495] = "path495.txt"
  [496] = "path496.txt"
  [497] = "path497.txt"
  [498] = "path498.txt"
  [499] = "path499.txt"
  [500] = "path500.txt"
string strCmd = "RBSTOP"
string strScrMsg[8]
  [1] = "F2===>move to ready"
  [2] = "F3===>points initial  "
  [3] = "F6===>test move"
  [4] = "F7===>TXT package initial"
  [5] = "F8===>exit"
string str_Dbg = "201.06"
tool tTip = {z=67.08, fatherId=flange[0], ioLink=valve1}
tool tTool = {z=125, fatherId=flange[0], ioLink=valve1}
trsf trsf_test
num n_Roate
num nRoateTotal

--- start.pgx ---
program start()
begin
  call initCmdBuf()
  call FC_InitData()
  waitEndMove()
  taskCreate "tcprec",100,TcpStrRec:SockRec(datar,ststu)
  call InitSocket()

  taskCreate "CmdManage",100,CmdManage()
  taskCreate "HMI",99,HMI()
  taskCreate "CmdDeal",99,CmdDealTest()
  taskCreate "CmdTxtReading",85,CmdTxtReading()
end

--- CmdDealTest.pgx ---
program CmdDealTest()
  local num l_ni
  local joint l_jTemp1
  local bool l_bTemp
begin


  while true



    if nReadPt!=nWritePt

      strCmd=mid(CmdBuffer[nReadPt],6,1)

      if strCmd=="RBREDY"

        popUpMsg("_")
        if bTxtPrSv==false
          popUpMsg("请首先对点位文件初始化（按F3-PoIn）")
        else
          //        // go to jCad[1] position

          //        //movej(jHome,tTool,mSlow)

          //        movej(jCad[1],tTool,mSlow)

          //        // movej(jReal,flange,mSlow)

          //        waitEndMove()

          //        //jConfig=herej()

          MoveTo.trsf=pfrmCad[0].trsf

          l_bTemp=pointToJoint(tTool,jConfig,MoveTo,l_jTemp1)

          //    $movejSync(jJointRx[l_nCount])

          l_jTemp1.j6=0
          movej(l_jTemp1,tTool,mNomSpeed)

          wait(isSettled()==true)

          socket="(RBREDY)"
        endIf

      endIf

      if strCmd=="RBSTOP"

        bSychronOn=false

        bRealM=false

        call FC_EndMotion()

        //        socket="(RBSTOP)"

        if taskStatus("SychMove")!=-1

          taskKill("SychMove")

          wait(taskStatus("SychMove")==-1)

        endIf

        if taskStatus("strToJt")!=-1

          taskKill("strToJt")

          wait(taskStatus("strToJt")==-1)

        endIf


        //
        call F4_DELT()
        call hmi_refreshmain()
      endIf


      //      if strCmd=="RBINIT"

      //        if nTotalPoints<=1

      //          //no point

      //          io:socket="(RBINIT)"

      //        else

      //          //delete points

      //          for l_ni=nTotalPoints to 2 step -1

      //            $ddel(jCad,nTotalPoints-1)

      //            nTotalPoints=nTotalPoints-1

      //            nScrPts=nTotalPoints

      //            call hmi_refreshmain()

      //          endFor

      //          wait(nTotalPoints==1)

      //          io:socket="(RBINIT)"

      //        endIf

      //      endIf

      if strCmd=="REALTM"

        //is realtime synchronous movement

        bRealM=true

      endIf

      if strCmd=="RBSTAT"
        if bTxtPrSv==false
          popUpMsg("请首先对点位文件初始化（按F3-PoIn）")
        else

          bfnshint=true

          //        if bfnshint==true

          //delay(0.0968)

          taskCreateSync "SychMove",0.004,bRes,task_sychron()

          //call task_sychron()

          //        else

          //          popUpMsg("init points frist")

          //          io:socket="(RBUNIN)"

          //        endIf
        endIf

      endIf

      CmdBuffer[nReadPt]=""

      CmdTotal=CmdTotal-1

      nReadPt=nReadPt+1

      if nReadPt>=20

        nReadPt=0

      endIf

    else

    endIf

    //delay(0)


  endWhile

end

--- CmdManage.pgx ---
program CmdManage()
begin
  while true
    if ststu==true and CmdTotal<20
      CmdBuffer[nWritePt]=datar
      CmdTotal=CmdTotal+1
      nWritePt=nWritePt+1
      if nWritePt>=20
        nWritePt=0
      endIf
      //HEREBELOW IS HIGH PRIORITY OF HOMING ROBOT
      datar=""
      ststu=false
    endIf
    delay(0)
  endWhile
end

--- CmdTxtReading.pgx ---
program CmdTxtReading()
begin
  //  call TxtHMI()
  //
  call Txt_initData()
  call Txt_PkgInit()
  nRoateTotal=5
  while true
   // if n_sTxt<nTxtTotal and nTxtTotal>2
   if n_Roate<nRoateTotal and nTxtTotal>2
      if bTxt1==true
        call TxtReadRoom1()
      else
      endIf
      if bTxt2==true
        call TxtReadRoom2()
      else
      endIf
      if bTxt3==true
        call TxtReadRoom3()
      else
      endIf
    else
    endIf
    //    nScrPts=n_sTxt
    //    call hmi_refreshmain()
  endWhile
end

--- DataSend2PC.pgx ---
program DataSend2PC()
  local num jold
  local bool bReconnect
begin
  //this routine is to send the data to PC
  while true
    delay(0)
  endWhile
end

--- F2_gohome.pgx ---
program F2_gohome()
  local joint l_jTemp1
  local bool l_bTemp
begin
  popUpMsg("ok")
  // go to pfrmCad[1] position
  if size(pfrmCad)>1
    //            //movej(jHome,tTool,mSlow)
    //            movej(jCad[1],flange,mSlow)
    MoveTo.trsf=pfrmCad[0].trsf
    l_bTemp=pointToJoint(tTool,jConfig,MoveTo,l_jTemp1)
    //    $movejSync(jJointRx[l_nCount])
    l_jTemp1.j6=0
    movej(l_jTemp1,tTool,mNomSpeed)
    waitEndMove()
  else
    popUpMsg("Motion need be initilized")
  endIf
end

--- F3_delete.pgx ---
program F3_delete()
  local num l_ni
begin
  //delete points
  //  nTotalPoints=size(pfrmCad)
  //  if nTotalPoints>1
  //    //      for l_ni=nTotalPoints to 2 step -1
  //    //        $ddel(pfrmCad,l_ni-1)
  //    ////        nTotalPoints=nTotalPoints-1
  //    ////        nScrPts=nTotalPoints
  //    //
  //    //      endFor
  //    //       call hmi_refreshmain()
  //    for l_ni=nTotalPoints to 2 step -1
  //      $ddel(pfrmCad,nTotalPoints-1)
  //      nTotalPoints=nTotalPoints-1
  //      nScrPts=nTotalPoints
  //    endFor
  //    call hmi_refreshmain()
  //  else
  //    popUpMsg("No points existed")
  //  endIf
end

--- F3_insertPs.pgx ---
public program F3_insertPs()
  local num l_nDbg
  local num j
  local num k
  local num l_n
  local bool l_bTemp
  local trsf l_trsf
  local joint l_jTemp1
begin
  //  //  call resetnum(nTest*(size(pTest)-1)+1)
  //  //  delay(0.2)
  //  //  for nDbg=0 to size(pTest)-2
  //  //    for nIONum=0 to nTest-1
  //  //      pCreatTest[nTest*nDbg+nIONum].trsf=interpolateL(pTest[nDbg].trsf,pTest[nDbg+1].trsf,nIONum/nTest)
  //  //
  //  //    endFor
  //  //  endFor
  //  //
  //  //  pCreatTest[nTest*(size(pTest)-1)].trsf=pTest[size(pTest)-1].trsf
  //  call resetnum(nPointnum)
  //  call partNum()
  //  delay(0.2)
  //  //jConfig=herej()
  //  //  for l_nDbg=0 to nPointnum-1
  //  //    cad:pCad[l_nDbg].trsf=interpolateC(pCircle[0].trsf,pCircle[1].trsf,pCircle[2].trsf,l_nDbg/(nPointnum-1))
  //  //    //MoveTo.trsf=position(cad:pCad[l_nDbg],FrmDraw)
  //  //    //l_bTemp=pointToJoint(tTool,jConfig,MoveTo,cad:jJointRx[l_nDbg])
  //  //  endFor
  //  l_n=0
  //  trsf_test={0,0,0,0,0,0}
  //  for j=0 to size(nPartNum)-1
  //    for k=0 to nPartNum[j]-1
  //      ptest.trsf=interpolateC(pCircle[2*j].trsf,pCircle[2*j+1].trsf,pCircle[2*j+2].trsf,k/(nPartNum[j]-1))
  //      //cad:pCad[l_n+k].trsf=interpolateC(pCircle[2*j].trsf,pCircle[2*j+1].trsf,pCircle[2*j+2].trsf,k/(nPartNum[j]-1))
  //      cad:pCad[l_n+k].trsf=position(ptest,FrmDraw)
  //      //////////test
  //      MoveTo.trsf=cad:pCad[l_n+k].trsf
  //      //坐标转换测试标记点。
  //      l_bTemp=pointToJoint(tTool,jConfig,MoveTo,cad:jJointRx[l_n+k])
  //      if l_n+k>0
  //        if abs(cad:pCad[l_n+k].trsf.x-cad:pCad[l_n+k-1].trsf.x)>trsf_test.x
  //          trsf_test.x=abs(cad:pCad[l_n+k].trsf.x-cad:pCad[l_n+k-1].trsf.x)
  //        endIf
  //        if abs(cad:pCad[l_n+k].trsf.y-cad:pCad[l_n+k-1].trsf.y)>trsf_test.y
  //          trsf_test.y=abs(cad:pCad[l_n+k].trsf.y-cad:pCad[l_n+k-1].trsf.y)
  //        endIf
  //        if abs(cad:pCad[l_n+k].trsf.z-cad:pCad[l_n+k-1].trsf.z)>trsf_test.z
  //          trsf_test.z=abs(cad:pCad[l_n+k].trsf.z-cad:pCad[l_n+k-1].trsf.z)
  //        endIf
  //        if abs(cad:pCad[l_n+k].trsf.rx-cad:pCad[l_n+k-1].trsf.rx)>trsf_test.rx
  //          trsf_test.rx=abs(cad:pCad[l_n+k].trsf.rx-cad:pCad[l_n+k-1].trsf.rx)
  //        endIf
  //        if abs(cad:pCad[l_n+k].trsf.ry-cad:pCad[l_n+k-1].trsf.ry)>trsf_test.ry
  //          trsf_test.x=abs(cad:pCad[l_n+k].trsf.x-cad:pCad[l_n+k-1].trsf.x)
  //        endIf
  //        if abs(cad:pCad[l_n+k].trsf.rz-cad:pCad[l_n+k-1].trsf.rz)>trsf_test.rz
  //          trsf_test.rz=abs(cad:pCad[l_n+k].trsf.rz-cad:pCad[l_n+k-1].trsf.rz)
  //        endIf
  //      endIf
  //      /////////
  //    endFor
  //    l_n=l_n+nPartNum[j]
  //  endFor
  //  cad:libSave()
  //  /////
  //  //  MoveTo.trsf=trsf_test
  //  //  l_bTemp=pointToJoint(tTool,jConfig,MoveTo,jTest)
  //  //////
  //  popUpMsg("OK")
end

--- F4_DELT.pgx ---
program F4_DELT()
begin
  //delay(10)
  delay(0.5)
  while size(sString)>1
    $ddel(sString,size(sString)-1)
  endWhile
  while size(nPulse)>1
    $ddel(nPulse,size(nPulse)-1)
  endWhile
  while size(pfrmCad)>1
    $ddel(pfrmCad,size(pfrmCad)-1)
  endWhile
  //sScrPts="NOT READY**"
  //bTxtPrSv=false
  bTxtPrSv=false
  sScrPts="NOT READY**"
  //n_sTxt=0
  n_sTxt=0
  call hmi_refreshmain()
end

--- F6_testmove.pgx ---
program F6_testmove()
  local num l_ni
  local bool l_bTemp
  local joint l_jTemp1
  local num l_nCount
begin
  //call FC_InitMotion()
  if bTxtPrSv==false
    popUpMsg("请首先对点位文件初始化（按F3-PoIn）")
  else
    pointToJoint(tTool,jConfig,pfrmCad[0],jConfig)
    MoveTo.trsf=pfrmCad[0].trsf
    l_bTemp=pointToJoint(tTool,jConfig,MoveTo,l_jTemp1)
    movej(l_jTemp1,tTool,mNomSpeed)
    l_nCount=0
    do
      if pfrmCad[l_nCount].trsf!={0,0,0,0,0,0}
        /////运动部分/////
        MoveTo.trsf=pfrmCad[l_nCount].trsf
        l_bTemp=pointToJoint(tTool,jConfig,MoveTo,l_jTemp1)
        movej(l_jTemp1,tTool,mNomSpeed)
        delay(0)
        /////运动部分/////
        pfrmCad[l_nCount].trsf={0,0,0,0,0,0}
        if l_nCount==600
          bTxt1=true
        endIf
        if l_nCount==1100
          bTxt2=true
        endIf
        if l_nCount==100
          bTxt3=true
        endIf
      endIf
      if l_nCount==1499
        l_nCount=0
      else
        l_nCount=l_nCount+1
      endIf
      delay(0)
    until pfrmCad[l_nCount].trsf=={0,0,0,0,0,0}
    bTxtPrSv=false
  endIf
  sScrPts="NotReady"
  call hmi_refreshmain()
  //
  //
  waitEndMove()
  popUpMsg("test over")
  //call FC_EndMotion()
end

--- F6_testsync.pgx ---
program F6_testsync()
begin
  //  if taskStatus("SychMove")==-1
  //    taskCreateSync "SychMove",0.004,bRes,task_sychron()
  //  endIf
end

--- FC_chrdeal.pgx ---
program FC_chrdeal(string& x_str[] (dimensions=1))
begin
  //delete all the space " "
  while left(x_str,1)==" "
    x_str=mid(x_str,len(x_str)-1,1)
  endWhile
end

--- FC_EndMotion.pgx ---
program FC_EndMotion()
begin
  //this function is to finish the synchronous motion
  $movejSyncEnd()
  //delay(5)
  //sScrPts="NOT READY"
  //n_sTxt=0
end

--- FC_InitData.pgx ---
program FC_InitData()
  local num l_ni
  local bool l_bInit
begin
  cls()
  userPage()
  // call hmi_keyinmain()
  bTxt1=false
  bTxt2=false
  bTxt3=false
end

--- FC_InitMotion.pgx ---
program FC_InitMotion()
begin
  //this function is goiong to begin the synchronous motion
  $movejSyncBegin(mNomSpeed)
end

--- hmi_keyinmain.pgx ---
program hmi_keyinmain()
  local num l_nKeyIn
  local num l_nDbg
  local num l_ni
begin
  //main page interface
  //clear message buffer
  cls()
  gotoxy(2,5)
  put("请输入txt文档总包数。如需修改，选择F7重新进行初始化")
  get(nTxtTotal)
  putln(nTxtTotal)
  sScrPts="NotReady"
  do
    l_nKeyIn=getKey()
    switch l_nKeyIn
      case 271
        //delete points
      break
      case 272
        // go to jCad[1] position
        call F2_gohome()
      break
      case 273
        call Txt_PkgInit()
      break
      case 274
        //         call Txt_PkgInit()
        call F4_DELT()
      break
      case 275
        call testMove()
      break
      case 276
        call F6_testmove()
      break
      case 277
        call hmi_keyinmain()
        //        call F7_testmove()
      break
      case 278
        //below is to confirm quit or not
        cls()
        gotoxy(2,5)
        put("Are you sure to quit ? 'Y' or ESC")
        l_nKeyIn=get()
        if l_nKeyIn==121
          l_nKeyIn=278
        else
          l_nKeyIn=0
        endIf
      break
    endSwitch
    //refresh hmi screen
    call hmi_refreshmain()
    //monitor production task ,if working mode in remote , start it automatically
  until (l_nKeyIn==278)
  //until ESC key is pushed
  //quite tasks and exit running staus
  //cls()
  //goto next page
end

--- hmi_refreshmain.pgx ---
program hmi_refreshmain()
begin
  //main page key input
  //  delay(0)
  cls()
  //put screen information
  title("SchronTest==>Slave")
  //event log display
  gotoxy(1,1)
  put("Menu operation───────────")
  gotoxy(1,2)
  put(strScrMsg[0])
  gotoxy(1,3)
  put(strScrMsg[1])
  gotoxy(1,4)
  put(strScrMsg[2])
  gotoxy(1,5)
  put(strScrMsg[3])
  gotoxy(1,6)
  put(strScrMsg[4])
  gotoxy(1,7)
  put(strScrMsg[5])
  gotoxy(1,8)
  put(strScrMsg[6])
  //  gotoxy(1,9)
  //  put(strScrMsg[7])
  gotoxy(1,9)
  put("Path Reading Num")
  gotoxy(23,9)
  put("      ")
  gotoxy(23,9)
  put(n_sTxt)
  gotoxy(1,10)
  put("TxtRoom")
  gotoxy(23,10)
  put("      ")
  gotoxy(23,10)
  put(sScrPts)
  gotoxy(1,11)
  put("TxtPKG Totals")

  gotoxy(23,11)
  put("      ")
  gotoxy(23,11)
  put(nTxtTotal)
  gotoxy(10,1)
  gotoxy(0,13)
  put("")
  gotoxy(5,13)
  put("RB2H")
  gotoxy(10,13)
  put("PoIn")
  gotoxy(15,13)
  put("DELT")
  gotoxy(20,13)
  put("TMOV")
  gotoxy(25,13)
  put("test")
  gotoxy(30,13)
  put("PkNm")
  gotoxy(35,13)
  put("Exit")
  //  gotoxy(0,13)
  //  put("RB1H")
  //  gotoxy(5,13)
  //  put("RB2H")
  //  gotoxy(10,13)
  //  put("PoIn")
  //  gotoxy(15,13)
  //  put("STOP")
  //  gotoxy(20,13)
  //  put("STAT")
  //  gotoxy(25,13)
  //  put("test ")
  //  gotoxy(30,13)
  //  put("TxIn ")
  //  gotoxy(35,13)
  //  put("Exit")
  delay(0.1)
  //recieve key and give actions
end

--- initCmdBuf.pgx ---
program initCmdBuf()
  local num i
begin
  for i=0 to 19
    CmdBuffer[i]=""
  endFor
  bfnshint=false
  CmdTotal=0
  nReadPt=0
  nWritePt=0
  setFrame(frm_ori,frm_x,frm_y,FrmDraw)
  MoveTo=Zero
  jConfig=jHome
  libSave()
end

--- InitSocket.pgx ---
public program InitSocket()
  local num l_nSocket
begin
  l_nSocket=clearBuffer(socket)
end

--- jCadClean.pgx ---
program jCadClean()
  local num l_ni
begin
  //  nTotalPoints=size(jCad)
  //  if nTotalPoints<=1
  //    //          //no point
  //    //          io:socket="(RBINIT)"
  //  else
  //    //delete points
  //    for l_ni=nTotalPoints to 2 step -1
  //      $ddel(jCad,nTotalPoints-1)
  //      nTotalPoints=nTotalPoints-1
  //      nScrPts=nTotalPoints
  //      call hmi_refreshmain()
  //    endFor
  //    wait(nTotalPoints==1)
  //    //          io:socket="(RBINIT)"
  //  endIf
end

--- partNum.pgx ---
program partNum()
  local num i
  local num l_n
  local num l_ndis
begin
  //  l_n=(size(pCircle)-1)/2
  //  while l_n<size(nPartdis)
  //    $ddel(nPartdis,size(nPartdis)-1)
  //    $ddel(nPartNum,size(nPartNum)-1)
  //  endWhile
  //  while l_n>size(nPartdis)
  //    $dins(nPartdis,size(nPartdis))
  //    $dins(nPartNum,size(nPartNum))
  //  endWhile
  //  for i=0 to l_n-1
  //    nPartdis[i]=distance(pCircle[2*i].trsf,pCircle[2*i+1].trsf)+distance(pCircle[2*i+2].trsf,pCircle[2*i+1].trsf)
  //    l_ndis=l_ndis+nPartdis[i]
  //  endFor
  //  for i=0 to l_n-1
  //    nPartNum[i]=round(nPointnum*nPartdis[i]/l_ndis)
  //  endFor
end

--- pFrmCadToJoint.pgx ---
program pFrmCadToJoint(pointRx x_pTemp (dimensions=1), joint& x_jTemp[] (dimensions=1))
  local num l_ni
  local bool l_bTemp
begin
  ////  if strCmd=="RBINIT"
  //
  ////  endIf
  //    l_bTemp=pointToJoint(tTool,jConfig,x_pPtemp,x_jTemp)
  //  if l_bTemp==false
  //    //    io:socket="(RBERRO)"
  //    popUpMsg("wrong point position!!!")
  //  endIf
end

--- PulesAdd.pgx ---
public program PulesAdd()
  local num l_nPulse
begin
  for l_nPulse=0 to 99 step 1
    delay(0.02)
    fOut0=true
    fOut0=false

  endFor

end

--- resetnum.pgx ---
program resetnum(num x_nNum1 (dimensions=1))
begin
  //  //  while size(pCreatTest)>x_nNum1
  //  //    $ddel(pCreatTest,size(pCreatTest)-1)
  //  //  endWhile
  //  //  while size(pCreatTest)<x_nNum1
  //  //    $dins(pCreatTest,size(pCreatTest))
  //  //  endWhile
  //  if x_nNum1>0
  //    while size(cad:pCad)>x_nNum1
  //      $ddel(cad:pCad,size(cad:pCad)-1)
  //      //$ddel(jJointRx,size(jJointRx)-1)
  //    endWhile
  //    while size(cad:jJointRx)>x_nNum1
  //      //$ddel(cad:pCad,size(cad:pCad)-1)
  //      $ddel(cad:jJointRx,size(cad:jJointRx)-1)
  //    endWhile
  //    while size(cad:jJointRx)<x_nNum1
  //      //$dins(cad:pCad,size(cad:pCad))
  //      $dins(cad:jJointRx,size(cad:jJointRx))
  //    endWhile
  //    while size(cad:pCad)<x_nNum1
  //      $dins(cad:pCad,size(cad:pCad))
  //      //$dins(jJointRx,size(jJointRx))
  //    endWhile
  //  else
  //    popUpMsg("点数应大于0")
  //  endIf
end

--- stop.pgx ---
program stop()
begin
  cls()
end

--- stringToJoints.pgx ---
program stringToJoints(string x_sStr (dimensions=1), joint& x_jTemp[] (dimensions=1))
  local string l_sX
  local string l_sY
  local num l_nPosX
  local num l_nPosY
  local bool l_bOk
  local num l_nPosZ
  local string l_sZ
  local bool l_bTemp
  local num l_ni
  local string l_sRX
  local string l_sRY
  local string l_sRZ
  local num l_nPosRX
  local num l_nPosRY
  local num l_nPosRZ
  local num l_nDbg
  local point l_ptest
begin
  //  l_sX=mid(x_sStr,7,13)
  //  call FC_chrdeal(l_sX)
  //  l_sY=mid(x_sStr,7,23)
  //  call FC_chrdeal(l_sY)
  //  l_sZ=mid(x_sStr,7,33)
  //  call FC_chrdeal(l_sZ)
  //  l_sRX=mid(x_sStr,7,43)
  //  call FC_chrdeal(l_sRX)
  //  l_sRY=mid(x_sStr,7,53)
  //  call FC_chrdeal(l_sRY)
  //  l_sRZ=mid(x_sStr,7,63)
  //  call FC_chrdeal(l_sRZ)
  //  toNum(l_sX,l_nPosX,l_bOk)
  //  toNum(l_sY,l_nPosY,l_bOk)
  //  toNum(l_sZ,l_nPosZ,l_bOk)
  //  toNum(l_sRX,l_nPosRX,l_bOk)
  //  toNum(l_sRY,l_nPosRY,l_bOk)
  //  toNum(l_sRZ,l_nPosRZ,l_bOk)
  //
  //  MoveTo.trsf.x=l_nPosX
  //  MoveTo.trsf.y=l_nPosY
  //  MoveTo.trsf.z=l_nPosZ
  //  MoveTo.trsf.rx=l_nPosRX
  //  MoveTo.trsf.ry=l_nPosRY
  //  MoveTo.trsf.rz=l_nPosRZ
  //  //MoveTo=position(l_ptest,FrmDraw)
  //  l_bTemp=pointToJoint(tTool,jConfig,MoveTo,x_jTemp)
  //  if l_bTemp==false
  //    io:socket="(RBERRO)"
  //    popUpMsg("wrong point position!!!")
  //  endIf
end

--- stringtopoint.pgx ---
program stringtopoint(string x_sString (dimensions=1), num x_nNum (dimensions=1))
  local string l_s
  local bool l_btest
  local num nX
  local num nY
  local num nZ
  local num nA
  local num nB
  local num nC
  local pointRx l_pPointRx
  local trsf tTrsf
  local pointRx pChangeMid1
  local num nP
  local pointRx pChangeMid2
begin
  l_s=x_sString
  l_s=toNum(l_s,nX,l_btest)
  l_s=toNum(l_s,nY,l_btest)
  l_s=toNum(l_s,nZ,l_btest)
  l_s=toNum(l_s,nA,l_btest)
  l_s=toNum(l_s,nB,l_btest)
  l_s=toNum(l_s,nC,l_btest)
  l_s=toNum(l_s,nP,l_btest)
  nPulse[x_nNum]=nP
  pChange.trsf.x=nX
  pChange.trsf.z=nZ
  pChange.trsf.y=nY
  ////  pChangeMid=compose(pChange,FrmDraw,{0,0,0,0,90,0})
  ////  pfrmCad[x_nNum]=compose(pChangeMid,FrmDraw,{0,0,0,0,0,nC})
  pChangeMid1=compose(pChange,FrmDraw,{0,0,0,nA,0,0})
  pChangeMid2=compose(pChangeMid1,FrmDraw,{0,0,0,0,0,nB})
  pfrmCad[x_nNum]=compose(pChangeMid2,FrmDraw,{0,0,0,nC,0,0})
  pfrmCad[x_nNum].trsf.x=pChange.trsf.x
  pfrmCad[x_nNum].trsf.z=pChange.trsf.z
  pfrmCad[x_nNum].trsf.y=pChange.trsf.y
  pChange[0].trsf={0,0,0,0,0,0}
end

--- sychronMove.pgx ---
public program sychronMove()
  local bool l_bTemp
  local num l_nCount
  local joint l_jTemp1
  local num l_nTime
begin
  //  //this task is synchronous moving
  //  //  MoveTo.trsf=cad:pCad[0].trsf
  //  //  l_bTemp=pointToJoint(tTool,jConfig,MoveTo,l_jTemp1)
  //  //  movej(l_jTemp1,tTool,mNomSpeed)
  //  //  waitEndMove()
  //  //  jConfig=herej()
  //  call FC_InitMotion()
  //  l_nCount=0
  //  bSetIO=true
  //  //
  //  nsumtime=clock()
  //  for l_nCount=0 to size(cad:pCad)-1
  //    //
  //    l_nTime=clock()
  //    //
  //    MoveTo.trsf=cad:pCad[l_nCount].trsf
  //    l_bTemp=pointToJoint(tTool,jConfig,MoveTo,l_jTemp1)
  //    $movejSync(l_jTemp1)
  //    //$movejSync(cad:jJointRx[l_nCount])
  //    l_nTime=clock()-l_nTime
  //    if l_nTime>nTime
  //      nTime=l_nTime
  //      nTestNum=l_nCount
  //    endIf
  //    delay(0)
  //  endFor
  //  //
  //  bSetIO=false
  //  //io:socket="(RBSTOP)"
  //  call FC_EndMotion()
  //  nsumtime=clock()-nsumtime
  //  popUpMsg("move end!")
  //  bTest=true
end

--- task_sychron.pgx ---
program task_sychron()
  local joint jTemp1
  local num l_ni
  local bool l_bTemp
  local num l_nCount
  local joint l_jTemp1
  local num l_nTime
begin
  //  call FC_InitMotion()
  //  call FC_InitMotion()
  //  //while true
  //  for l_ni=1 to size(jCad)-1
  //    $movejSync(jCad[l_ni])
  //    delay(0)
  //  endFor
  //  call FC_EndMotion()
  nn=0
  call FC_InitMotion()
  l_nCount=0
  n_Roate=0
  bSetIO=true
  nRoateTotal=5
  nsumtime=clock()
  do
    if pfrmCad[l_nCount].trsf!={0,0,0,0,0,0}
      //////替换
      //  for l_nCount=1 to size(pfrmCad)-1
      //
      l_nTime=clock()
      MoveTo.trsf=pfrmCad[l_nCount].trsf
      l_bTemp=pointToJoint(tTool,jConfig,MoveTo,l_jTemp1)
      l_jTemp1.j6=0
      $movejSync(l_jTemp1)
      if nPulse[l_nCount]==1
        fOut0=true
        fOut0=false
        nn=nn+1
      else
      endIf
      /////运动部分/////
      pfrmCad[l_nCount].trsf={0,0,0,0,0,0}
      if l_nCount==600
        bTxt1=true
      endIf
      if l_nCount==1100
        bTxt2=true
      endIf
      if l_nCount==100
        bTxt3=true
      endIf
    endIf
    if l_nCount==1499
      l_nCount=0
    else
      l_nCount=l_nCount+1
    endIf
    //    delay(0)
    l_nTime=clock()-l_nTime
    if l_nTime>nTime
      nTime=l_nTime
      nTestNum=l_nCount
    endIf
    delay(0)
  until pfrmCad[l_nCount].trsf=={0,0,0,0,0,0}

  do
    if l_nCount>0 and l_nCount<500
      l_nCount=500
    endIf

    if 500<l_nCount and l_nCount<1000
      l_nCount=1000
    endIf

    if 1000<l_nCount and l_nCount<1500
      l_nCount=0
    endIf

    do
      if pfrmCad[l_nCount].trsf!={0,0,0,0,0,0}
        //////替换
        //  for l_nCount=1 to size(pfrmCad)-1
        //
        l_nTime=clock()
        MoveTo.trsf=pfrmCad[l_nCount].trsf
        l_bTemp=pointToJoint(tTool,jConfig,MoveTo,l_jTemp1)
        l_jTemp1.j6=0
        $movejSync(l_jTemp1)
        if nPulse[l_nCount]==1
          fOut0=true
          fOut0=false
          nn=nn+1
        else
        endIf
        /////运动部分/////
        pfrmCad[l_nCount].trsf={0,0,0,0,0,0}
        if l_nCount==600
          bTxt1=true
        endIf
        if l_nCount==1100
          bTxt2=true
        endIf
        if l_nCount==100
          bTxt3=true
        endIf
      endIf
      if l_nCount==1499
        l_nCount=0
      else
        l_nCount=l_nCount+1
      endIf
      //    delay(0)
      l_nTime=clock()-l_nTime
      if l_nTime>nTime
        nTime=l_nTime
        nTestNum=l_nCount
      endIf
      delay(0)
    until pfrmCad[l_nCount].trsf=={0,0,0,0,0,0}

    n_Roate=n_Roate+1
  until n_Roate==nRoateTotal-1

  delay(1)

  while size(sString)>1
    $ddel(sString,size(sString)-1)
  endWhile
  while size(nPulse)>1
    $ddel(nPulse,size(nPulse)-1)
  endWhile
  while size(pfrmCad)>1
    $ddel(pfrmCad,size(pfrmCad)-1)
  endWhile
  delay(0)

  call PulesAdd()

  bTxt1=false
  bTxt2=false
  bTxt3=false
  //    //
  //    //    MoveTo.trsf=cad:pCad[l_nCount].trsf
  //    //    l_bTemp=pointToJoint(tTool,jConfig,MoveTo,l_jTemp1)
  //    //    $movejSync(jCad[l_nCount])
  //    MoveTo.trsf=pfrmCad[l_nCount].trsf
  //    l_bTemp=pointToJoint(tTool,jConfig,MoveTo,l_jTemp1)
  //    $movejSync(l_jTemp1)
  //    //$movejSync(cad:jJointRx[l_nCount])
  //    l_nTime=clock()-l_nTime
  //    if l_nTime>nTime
  //      nTime=l_nTime
  //      nTestNum=l_nCount
  //    endIf
  //    delay(0)
  //  endFor
  /////替换/
  //  for l_nCount=0 to size(cad:pCad)-1
  //    //
  //    l_nTime=clock()
  //    //
  //    MoveTo.trsf=cad:pCad[l_nCount].trsf
  //    l_bTemp=pointToJoint(tTool,jConfig,MoveTo,l_jTemp1)
  //    $movejSync(l_jTemp1)
  //    //$movejSync(cad:jJointRx[l_nCount])
  //    l_nTime=clock()-l_nTime
  //    if l_nTime>nTime
  //      nTime=l_nTime
  //      nTestNum=l_nCount
  //    endIf
  //    delay(0)
  //  endFor
  ///////替换
  bSetIO=false
  //io:socket="(RBSTOP)"
  call FC_EndMotion()
  nsumtime=clock()-nsumtime
  bTxtPrSv=false
  sScrPts="NotReady"
  n_sTxt=0
  call hmi_refreshmain()
  //popUpMsg("move end!")
  bTest=true
end

--- testMove.pgx ---
program testMove()
begin
  bfnshint=true
  //        if bfnshint==true
  //delay(0.0968)
  taskCreateSync "SychMove",0.004,bRes,task_sychron()
  //call task_sychron()
end

--- Txt_initData.pgx ---
program Txt_initData()
  local num l_nInit
begin
  //    title("Please Enter Txt Files Total number")
  //  cls()
  //  popUpMsg("请在点击OK后输入txt文档总包数（显示在左下角），并点回车。如需修改，选择F7重新进行初始化")
  //  get(nTxtTotal)
  //  putln(nTxtTotal)
  //  call Txt_initData()
  while size(sString)>1
    $ddel(sString,size(sString)-1)
  endWhile
  while size(nPulse)>1
    $ddel(nPulse,size(nPulse)-1)
  endWhile
  while size(pfrmCad)>1
    $ddel(pfrmCad,size(pfrmCad)-1)
  endWhile
  pfrmCad[0].trsf={0,0,0,0,0,0}
  sString[0]=""
  for l_nInit=1 to 1499
    $dins(sString,l_nInit)
    $dins(nPulse,l_nInit)
    $dins(pfrmCad,l_nInit)
  endFor
  bTxtPrSv=false
  //  popUpMsg("txt is ready")
end

--- Txt_PkgInit.pgx ---
program Txt_PkgInit()
begin
  n_sTxt=0
  call Txt_initData()
  call TxtReadRoom1()
  if nTxtTotal>1
    call TxtReadRoom2()
  endIf
  bTxtPrSv=true
  sScrPts="OK"
  call hmi_refreshmain()
end

--- txt_rd.pgx ---
public program txt_rd()
  local num l_ntest
  local num l_n
  local num l_mark
begin
  //  l_ntest=$fileOpen("test2.txt","r")
  //  //  直接更改数量，注意point及sstring要与其一致
  //  //  for l_n=0 to 1
  //  //    $fileGet(l_ntest,sString[l_n],1)
  //  //    if sString[l_n]!=""
  //  //      call stringtopoint(sString[l_n],l_n)
  //  //    endIf
  //  //  endFor
  //  ///////初始化
  //  l_n=0
  //  while size(sString)>1
  //    $ddel(sString,size(sString)-1)
  //  endWhile
  //  while size(pfrmCad)>1
  //    $ddel(pfrmCad,size(pfrmCad)-1)
  //  endWhile
  //  ///////////////
  //  do
  //    if l_n!=0
  //      $dins(sString,l_n)
  //      $dins(pfrmCad,l_n)
  //    endIf
  //    $fileGet(l_ntest,sString[l_n],1)
  //    if sString[l_n]!=""
  //      call stringtopoint(sString[l_n],l_n)
  //    else
  //    endIf
  //    l_n=l_n+1
  //  until sString[l_n-1]==""
  //  $ddel(sString,size(sString)-1)
  //  $ddel(pfrmCad,size(pfrmCad)-1)
  //  delay(0.1)
  //  $fileClose(l_ntest)
  //  //读取参考系中的点
  //  call jCadClean()
  //  //清空jcad
  //  for l_mark=0 to size(pfrmCad)-1 step 1
  //    pointToJoint(tTool,jConfig,pfrmCad[l_mark],jReal)
  //    nTotalPoints=nTotalPoints+1
  //    $dins(jCad,nTotalPoints-1)
  //    jCad[nTotalPoints-1]=jReal
  //    nScrPts=nTotalPoints
  //    delay(0)
  //
  //
  //  endFor
  //  bfnshint=true
  //  //将pfrmcad逐个转化成jcad的joint点。
  //  /////////////////////////////////////
  //  /////////////////////////////////////
  ////        call stringToJoints(CmdBuffer[nReadPt],jReal)
  ////        if bRealM==true
  ////          //for realtime synchronous movement
  ////        else
  ////          //for initialize all points firstly
  ////          //not realtime synchronous movement
  ////          nTotalPoints=nTotalPoints+1
  ////          $dins(jCad,nTotalPoints-1)
  ////          jCad[nTotalPoints-1]=jReal
  ////
  ////          nScrPts=nTotalPoints
  ////          call hmi_refreshmain()
  ////        endIf
  ////      endIf
end

--- txt_rd1.pgx ---
public program txt_rd1()
  local num l_ntest
  local num l_n
  local num l_mark
  local bool l_jtest
begin
  //  l_ntest=$fileOpen("test.txt","r")
  //  //  直接更改数量，注意point及sstring要与其一致
  //  //  for l_n=0 to 1
  //  //    $fileGet(l_ntest,sString[l_n],1)
  //  //    if sString[l_n]!=""
  //  //      call stringtopoint(sString[l_n],l_n)
  //  //    endIf
  //  //  endFor
  //  ///////初始化
  //  l_n=0
  //  //  while size(sString)>1
  //  //    $ddel(sString,size(sString)-1)
  //  //  endWhile
  //  //  while size(pfrmCad)>1
  //  //    $ddel(pfrmCad,size(pfrmCad)-1)
  //  //  endWhile
  //  //  while size(jCad)>1
  //  //    $ddel(jCad,size(jCad)-1)
  //  //  endWhile
  //  ///////////////
  //  //  popUpMsg("已经开始读点，请稍等...")
  //  do
  //    if l_n!=0
  //      $dins(sString,l_n)
  //      $dins(pfrmCad,l_n)
  //    endIf
  //    $fileGet(l_ntest,sString[l_n],1)
  //    if sString[l_n]!=""
  //      call stringtopoint(sString[l_n],l_n)
  //    else
  //    endIf
  //    l_n=l_n+1
  //  until sString[l_n-1]==""
  //  $ddel(sString,size(sString)-1)
  //  $ddel(pfrmCad,size(pfrmCad)-1)
  //  delay(0.1)
  //  nScrPts=size(pfrmCad)
  //  call hmi_refreshmain()
  //  popUpMsg("读取完毕")
  //  $fileClose(l_ntest)
  //  //读取参考系中的点
  //  //  call jCadClean()
  //  //清空jcad
  //  //  nTotalPoints=size(pfrmCad)
  //  //  for l_mark=1 to nTotalPoints-1 step 1
  //  //    $dins(jCad,l_mark)
  //  //  endFor
  //  //  for l_mark=0 to size(pfrmCad)-1 step 1
  //  //    l_jtest=pointToJoint(tTool,jConfig,pfrmCad[l_mark],jReal)
  //  //    if l_jtest==false
  //  //      popUpMsg("point is wrong")
  //  //      return
  //  //    else
  //  //      jCad[l_mark]=jReal
  //  //      // jCad[nTotalPoints-1]=jHome
  //  //      //      $dins(jCad,nTotalPoints)
  //  //      ////      nScrPts=nTotalPoints
  //  //      //      nTotalPoints=nTotalPoints+1
  //  //      delay(0)
  //  //    endIf
  //  //  endFor
  //  //   $ddel(jCad,size(jCad))
  //  bfnshint=true
  //  //将pfrmcad逐个转化成jcad的joint点。
  //  /////////////////////////////////////
  //  /////////////////////////////////////
  //  //        call stringToJoints(CmdBuffer[nReadPt],jReal)
  //  //        if bRealM==true
  //  //          //for realtime synchronous movement
  //  //        else
  //  //          //for initialize all points firstly
  //  //          //not realtime synchronous movement
  //  //          nTotalPoints=nTotalPoints+1
  //  //          $dins(jCad,nTotalPoints-1)
  //  //          jCad[nTotalPoints-1]=jReal
  //  //
  //  //          nScrPts=nTotalPoints
  //  //          call hmi_refreshmain()
  //  //        endIf
  //  //      endIf
end

--- TxtReadRoom1.pgx ---
program TxtReadRoom1()
  local num l_ntest
  local num l_n
begin
  delay(0.01)
  l_ntest=$fileOpen(sTxtfile[n_sTxt],"r")
  for l_n=0 to 499
    $fileGet(l_ntest,sString[l_n],1)
    if sString[l_n]!=""
      call stringtopoint(sString[l_n],l_n)
    else
    endIf
  endFor
  delay(0.01)
  bTxt1=false
  if n_sTxt==nTxtTotal-1
    n_sTxt=0
  else
    n_sTxt=n_sTxt+1
  endIf

  $fileClose(l_ntest)
  call hmi_refreshmain()
end

--- TxtReadRoom2.pgx ---
program TxtReadRoom2()
  local num l_ntest
  local num l_n
begin
  delay(0.01)
  l_ntest=$fileOpen(sTxtfile[n_sTxt],"r")
  for l_n=500 to 999
    $fileGet(l_ntest,sString[l_n],1)
    if sString[l_n]!=""
      call stringtopoint(sString[l_n],l_n)
    else
    endIf
  endFor
  delay(0.01)
  bTxt2=false
 if n_sTxt==nTxtTotal-1
  n_sTxt=0
else
  n_sTxt=n_sTxt+1
endIf

  $fileClose(l_ntest)
  call hmi_refreshmain()
end

--- TxtReadRoom3.pgx ---
program TxtReadRoom3()
  local num l_ntest
  local num l_n
begin
  delay(0.01)
  l_ntest=$fileOpen(sTxtfile[n_sTxt],"r")
  for l_n=1000 to 1499
    $fileGet(l_ntest,sString[l_n],1)
    if sString[l_n]!=""
      call stringtopoint(sString[l_n],l_n)
    else
    endIf
  endFor
  delay(0.01)
  bTxt3=false
  if n_sTxt==nTxtTotal-1
    n_sTxt=0
  else
    n_sTxt=n_sTxt+1
  endIf

  $fileClose(l_ntest)
  call hmi_refreshmain()
end
